(* POU PRG_STATION_LAYER3/FB_STATIONEN/FB_FUNCTION/FB_STATION, ST *)
FUNCTION_BLOCK FB_STATION
VAR_INPUT
	iConfigMachineType:INT;
	iConfigAxisType:INT;
	iConfigVisuNavigation:INT;
	rConfigMaxToolLength:REAL;
	xSafetyCircuitOn1:BOOL;
	xSafetyCircuitOn2:BOOL;
	T_ProcessImageData:ST_RETAIN_DATA_PROCESSIMAGE;
	T_Standard:ST_RETAIN_DATA;
	xActiveProcess:BOOL;
	iSelectToolTensionForce:INT;
END_VAR
VAR_IN_OUT
	TStation:ST_STATION;
	T_StartUp:ST_STARTUP;
END_VAR
VAR_OUTPUT
	xActive : BOOL :=FALSE;
	xStatusRdy : BOOL := FALSE;
	xStatusEnd : BOOL := FALSE;
	xStatusStop : BOOL := FALSE;
	xStatusRef : BOOL := FALSE;
	xError : BOOL := FALSE;
	iErrorNr : DINT :=0;
	iStatusFctNr : INT := 0;
	bActivePartNumber:BYTE;
	lrProcessToolFeederActualPosition:LREAL;
	lrProcessToolFeederSpeed:LREAL;
END_VAR
VAR
(* Pointer auf Actuatoren *)
	ptrTAxisToolLeft:POINTER TO ST_AXIS;
	ptrTAxisToolCenter:POINTER TO ST_AXIS;
	ptrTAxisToolRight:POINTER TO ST_AXIS;
	ptrTAxisToolFeeder:POINTER TO ST_AXIS;
	ptrTAxisGrindFeeder:POINTER TO ST_AXIS;
	ptrTCylToolTension:POINTER TO ST_CYLINDER;
(*22.12.2009: KFS {    *)
	ptrTCylToolLeftActive:POINTER TO ST_CYLINDER;
	ptrTCylToolRightActive:POINTER TO ST_CYLINDER;
	ptrTCylToolCenterActive:POINTER TO ST_CYLINDER;
	ptrTCylToolPrismaLeftActive:POINTER TO ST_CYLINDER;
	ptrTCylToolPrismaRightActive:POINTER TO ST_CYLINDER;
	ptrTToolFeederWorkLength:POINTER TO ST_CYLINDER;
(*22.12.2009: KFS }   *)
	ptrTFunction:POINTER TO ST_CTRL_FUNCTION;
	xSetEnableConfig: BOOL;
	iEnableConfigMachineType:INT;
	iTmpConfigMachineType:INT;
	iEnableConfigAxisType:INT;
	iTmpConfigAxisType:INT;
	iEnableConfigVisuNavigation:INT;
	iTmpConfigVisuNavigation:INT;
	rEnableConfigMaxToolLength:REAL;
	rTmpConfigMaxToolLength:REAL;
	xMicroRodActive: BOOL;
	xBeckhoffDriveActive: BOOL;
	xTmpStopFunction: BOOL;
	iStationFunctionNr: INT;
	xStartFunction: BOOL := FALSE;
	xTmpStart: BOOL := FALSE;
	xInitStart: BOOL := FALSE;
	xSetEnd: BOOL := FALSE;
	xInitError: BOOL := FALSE;
	xInitStop: BOOL := FALSE;
	xInitSetEnable: BOOL := FALSE;
	iStepEnable: INT := 0;
	xInitStep: BOOL := FALSE;
	iAxisFunctionNr: INT :=0;
	xInitDelEnable: BOOL := FALSE;
	xStationError: BOOL := FALSE;
	xStepError: BOOL;
	iStepError: INT;
	xTmpStationError: BOOL;
	xRdyDisableStation: BOOL;
	xReadyChkError: BOOL;
	xDontDeleteErrorFlag: BOOL;
	xSetError: BOOL;
(* Trigger *)
	fbFTrig: F_TRIG;
	fbRTrig: R_TRIG;
	xTmp: BOOL;
	diErrorNumber: DINT;
	iCountCycle: INT;
	xSecurityCircuitOn: BOOL;
	xSecurityCircuitOff: BOOL;
	iStepSecCircuit: INT;
	xInitSecCircuit: BOOL;
	TONCheckTimeOut: TON;
	xPowerSwitchedOn: BOOL;
	xChkConfigStation: BOOL;
	FBFctToolRotationTorqueStart: FB_FctToolRotationTorqueStart;
	FBFctToolRotationTorqueStop: FB_FctToolRotationTorqueStop;
	FBFctGrindFeedAbsRelPosition: FB_FctGrindFeedAbsRelPosition;
	FBFctSetAxisPosition: FB_FctSetAxisPosition;
	FBFctToolWorkingGeometry: FB_FctToolWorkingGeometry;
	FBFctToolWorkingGeometryMultiCycle: FB_FctToolWorkingGeometryMultiCycle;
	FBFctToolWorkingGroove: FB_FctToolWorkingGroove;
	FBFctToolCalibration: FB_FctToolCalibration;
	iMaxFunctionNr:INT:=20;
	(* 17.11.2010 KFS : iMaxFunctionNr:INT:=19*)
	FBFctToolFeedAbsRelPosition: FB_FctToolFeedAbsRelPosition;
	FBFctSwitchOnOffPowerSupply: FB_FctSwitchOnOffPowerSupply;
	(* 17.11.2010: KFS 	{	*)
	FBFctToolFeedMaxLenReference:FB_FctToolFeedMaxLenReference;
	(* 17.11.2010: KFS 	}	*)
	FBFctToolFeedReference: FB_FctToolFeedReference;
	xCheckAxisError: BOOL;
	xFirstTimeBooting: BOOL:=FALSE;
	FBFctStopAxisMovement: FB_FctStopAxisMovement;
	xAxisErrorActive: BOOL;
	xWaitSetError: BOOL;
	TONWaitSetError: TON;
	xForceHWError: BOOL;
	xCheckActiveFunction: BOOL;
	xForceResetAxis: BOOL;
	xReadyToQuitErr: BOOL;
	TONWaitReset: TON;
END_VAR
(****************************************************************************************************************************************************)
(***********                 This Functionblock manage all the station funtion and synchronizing of the Hardware                           ************)
(****************************************************************************************************************************************************)
xActive:=TStation.TControl.xActiveStation;
IF NOT(TStation.TControl.xActiveStation) THEN
	(*TStation:=TDeleteStationStruct;*)
	RETURN;
ELSE
	IF xSetEnableConfig THEN
		IF (iEnableConfigMachineType <> iConfigMachineType) THEN
			iTmpConfigMachineType:=iEnableConfigMachineType;
		ELSE
			iTmpConfigMachineType:=iConfigMachineType;
		END_IF;
		IF (iEnableConfigAxisType <> iConfigAxisType) THEN
			iTmpConfigAxisType:=iEnableConfigAxisType;
		ELSE
			iTmpConfigAxisType:=iConfigAxisType;
		END_IF;
		IF (iEnableConfigVisuNavigation <> iConfigVisuNavigation) THEN
			iTmpConfigVisuNavigation:=iEnableConfigVisuNavigation;
		ELSE
			iTmpConfigVisuNavigation:=iConfigVisuNavigation;
		END_IF;
		IF (rEnableConfigMaxToolLength <> rConfigMaxToolLength) THEN
			rTmpConfigMaxToolLength:=rEnableConfigMaxToolLength;
		ELSE
			rTmpConfigMaxToolLength:=rConfigMaxToolLength;
		END_IF;
		(*08.12.2010 KFS:	{	*)
		IF T_Station.xOverwriteMaxToolLength THEN
			rEnableConfigMaxToolLength:=rConfigMaxToolLength;
			rTmpConfigMaxToolLength:=rConfigMaxToolLength;
		END_IF;
		(*08.12.2010 KFS:	}	*)
	ELSE
		iTmpConfigMachineType:=iConfigMachineType;
		iTmpConfigAxisType:=iConfigAxisType;
		iTmpConfigVisuNavigation:=iConfigVisuNavigation;
		rTmpConfigMaxToolLength:=rConfigMaxToolLength;
	END_IF;
	(* Zuweisung der Datenstrukturen der Aktuatoren als Pointer *)
	ptrTAxisToolLeft:=ADR(TStation.THardware.TAxisToolLeft);
	ptrTAxisToolCenter:=ADR(TStation.THardware.TAxisToolCenter);
	ptrTAxisToolRight:=ADR(TStation.THardware.TAxisToolRight);
	ptrTAxisToolFeeder:=ADR(TStation.THardware.TAxisToolFeeder);
	ptrTAxisGrindFeeder:=ADR(TStation.THardware.TAxisGrindFeeder);
	ptrTCylToolTension:=ADR(TStation.THardware.TCylToolTension);
(*22.12.2009: KFS {    *)
	ptrTCylToolLeftActive:=ADR(TStation.THardware.TCylToolLeftActive);
	ptrTCylToolRightActive:=ADR(TStation.THardware.TCylToolRightActive);
	ptrTCylToolCenterActive:=ADR(TStation.THardware.TCylToolCenterActive);
	ptrTCylToolPrismaLeftActive:=ADR(TStation.THardware.TCylToolPrismaLeftActive);
	ptrTCylToolPrismaRightActive:=ADR(TStation.THardware.TCylToolPrismaRightActive);
	ptrTToolFeederWorkLength:=ADR(TStation.THardware.TToolFeederWorkLength);
(*22.12.2009: KFS }   *)
	ptrTFunction:=ADR(TStation.TCtrlFunction);
	IF (iConfigMachineType = 2) THEN
		xMicroRodActive:=TRUE;
	ELSE
		xMicroRodActive:=FALSE;
	END_IF;
	IF (iConfigAxisType = 2) THEN
		xBeckhoffDriveActive:=TRUE;
	ELSE
		xBeckhoffDriveActive:=FALSE;
	END_IF;
	IF xSafetyCircuitOn1 AND xSafetyCircuitOn2 THEN
		xPowerSwitchedOn:=TRUE;
	ELSE
		xPowerSwitchedOn:=FALSE;
	END_IF;
END_IF;
(******************************************************************************************************************************************)
(****************************				                  Status Part                                                            *****************************)
(******************************************************************************************************************************************)
xStatusRdy:=TStation.TControl.xRdy;
xStatusEnd:=TStation.TControl.xEnd;
xStatusStop:=xTmpStopFunction;
IF xMicroRodActive THEN
	TStation.TControl.xReferenced:=ptrTAxisToolFeeder^.T_CtrleSingle.xRef;
ELSE
	TStation.TControl.xReferenced:=TRUE;
END_IF;
xStatusRef:=TStation.TControl.xReferenced;
xError:= TStation.TControl.xError;
iErrorNr := TStation.TControl.diErrorNr;
iStatusFctNr:=iStationFunctionNr;
(******************************************************************************************************************************************)
(****************************				                Enable Part                                                            *****************************)
(******************************************************************************************************************************************)
(* Check Active of the Axis Drives *)
xTmp:=	(NOT(ptrTAxisToolLeft^.T_CtrleSingle.xErr) AND NOT(ptrTAxisToolLeft^.T_CtrleSingle.xDone)) OR
		(NOT(ptrTAxisToolCenter^.T_CtrleSingle.xErr) AND NOT(ptrTAxisToolCenter^.T_CtrleSingle.xDone) AND xMicroRodActive) OR
		(NOT(ptrTAxisToolRight^.T_CtrleSingle.xErr) AND NOT(ptrTAxisToolRight^.T_CtrleSingle.xDone)) OR
		(NOT(ptrTAxisToolFeeder^.T_CtrleSingle.xErr) AND NOT(ptrTAxisToolFeeder^.T_CtrleSingle.xDone)) OR
		(NOT(ptrTAxisGrindFeeder^.T_CtrleSingle.xErr) AND NOT(ptrTAxisGrindFeeder^.T_CtrleSingle.xDone));
fbFTrig(CLK:=TStation.TControl.xEnable);
IF fbFTrig.Q THEN
	xInitSetEnable:=FALSE;
	xInitDelEnable:=FALSE;
	xRdyDisableStation:=FALSE;
END_IF;
IF (fbFTrig.Q OR xInitDelEnable) THEN
	IF NOT(xInitDelEnable) OR fbFTrig.Q THEN
		xReadyChkError:=FALSE;
		TStation.TControl.xEnd:=FALSE;
		IF NOT(xDontDeleteErrorFlag) THEN
			TStation.TControl.xError:=FALSE;
		END_IF;
		xInitDelEnable:=TRUE;
		TStation.TControl.xRdy:=FALSE;
		iStepEnable:=100;
		iAxisFunctionNr:=1;
		iStationFunctionNr:=1;
		xInitStep:=FALSE;
	END_IF;
	CASE iStepEnable OF
		100:	IF NOT(xInitStep) THEN
				xInitStep:=TRUE;
				xSetEnableConfig:=FALSE;
				xStartFunction:=TRUE;
				ptrTFunction^.xReset:=TRUE;
			END_IF;
			IF NOT(ptrTFunction^.xReset) AND ptrTFunction^.xEnd THEN
				(* Alle Funktionen Resetten *)
				IF (iStationFunctionNr < iMaxFunctionNr) THEN
					iStationFunctionNr:=iStationFunctionNr + 1;
					ptrTFunction^.xReset:=TRUE;
				ELSE
					xInitStep:=FALSE;
					xStartFunction:=FALSE;
					iStepEnable:=200;
				END_IF;
			END_IF;
		200:	IF NOT(xInitStep) THEN
				xInitStep:=TRUE;
				IF TStation.TControl.xHardwareConfigError THEN
					TStation.TControl.xHardwareConfigError:=FALSE;
					TStation.TControl.xActiveHardware:=FALSE;
				ELSE
					xInitStep:=FALSE;
					iStepEnable:=300;
				END_IF;
				RETURN;
			END_IF;
			IF NOT(TStation.TControl.xError) OR xDontDeleteErrorFlag THEN
				TStation.TControl.xActiveHardware:=TRUE;
				xInitStep:=FALSE;
				iStepEnable:=300;
				RETURN;
			END_IF;
		300:	IF NOT(xInitStep) THEN	(* Alle Hardware Bausteine resetten *)
				xInitStep:=TRUE;
				ptrTCylToolTension^.T_CtrleCyl.xFBActiv:=FALSE;
				(*22.12.2009: KFS {    *)
				IF xMicroRodActive THEN
					ptrTCylToolLeftActive^.T_CtrleCyl.xFBActiv:=FALSE;
					ptrTCylToolRightActive^.T_CtrleCyl.xFBActiv:=FALSE;
					ptrTCylToolCenterActive^.T_CtrleCyl.xFBActiv:=FALSE;
					ptrTCylToolPrismaLeftActive^.T_CtrleCyl.xFBActiv:=FALSE;
					ptrTCylToolPrismaRightActive^.T_CtrleCyl.xFBActiv:=FALSE;
					ptrTToolFeederWorkLength^.T_CtrleCyl.xFBActiv:=FALSE;
				END_IF;
				(*22.12.2009: KFS }   *)
				IF xBeckhoffDriveActive THEN
					ptrTAxisToolLeft^.T_CtrleSingle.xReset:=TRUE;
					IF xMicroRodActive THEN
						ptrTAxisToolCenter^.T_CtrleSingle.xReset:=TRUE;
					END_IF;
					ptrTAxisToolRight^.T_CtrleSingle.xReset:=TRUE;
					ptrTAxisToolFeeder^.T_CtrleSingle.xReset:=TRUE;
					ptrTAxisGrindFeeder^.T_CtrleSingle.xReset:=TRUE;
				ELSE
					TStation.TControl.xResetHardware:=TRUE;
					iStepEnable:=399;
					RETURN;
				END_IF;
			END_IF;
			IF xTmp THEN
				RETURN;	(* Wait until all Drives finished *)
			END_IF;
			IF (NOT(ptrTAxisToolLeft^.T_CtrleSingle.xReset) AND ptrTAxisToolLeft^.T_CtrleSingle.xErr) OR
			    (((NOT(ptrTAxisToolCenter^.T_CtrleSingle.xReset) AND ptrTAxisToolCenter^.T_CtrleSingle.xErr AND xMicroRodActive) OR NOT(xMicroRodActive))) OR
			    (NOT(ptrTAxisToolRight^.T_CtrleSingle.xReset) AND ptrTAxisToolRight^.T_CtrleSingle.xErr) OR
			    (NOT(ptrTAxisToolFeeder^.T_CtrleSingle.xReset) AND ptrTAxisToolFeeder^.T_CtrleSingle.xErr)OR
			    (NOT(ptrTAxisGrindFeeder^.T_CtrleSingle.xReset) AND ptrTAxisGrindFeeder^.T_CtrleSingle.xErr) THEN
				xInitStep:=FALSE;
				iStepEnable:=400;
			END_IF;
			IF NOT(ptrTAxisToolLeft^.T_CtrleSingle.xReset) AND ptrTAxisToolLeft^.T_CtrleSingle.xDone AND
			    ((NOT(ptrTAxisToolCenter^.T_CtrleSingle.xReset) AND ptrTAxisToolCenter^.T_CtrleSingle.xDone AND xMicroRodActive) OR NOT(xMicroRodActive)) AND
			    NOT(ptrTAxisToolRight^.T_CtrleSingle.xReset) AND ptrTAxisToolRight^.T_CtrleSingle.xDone AND
			    NOT(ptrTAxisToolFeeder^.T_CtrleSingle.xReset) AND ptrTAxisToolFeeder^.T_CtrleSingle.xDone AND
			    NOT(ptrTAxisGrindFeeder^.T_CtrleSingle.xReset) AND ptrTAxisGrindFeeder^.T_CtrleSingle.xDone THEN
				TStation.TControl.xActiveHardware:=FALSE;
				xInitStep:=FALSE;
				xInitDelEnable:=FALSE;
				xSetEnd:=TRUE;
				xRdyDisableStation:=TRUE;
			END_IF;
		399:	IF NOT(TStation.TControl.xResetHardware) THEN
				TStation.TControl.xActiveHardware:=FALSE;
				xInitStep:=FALSE;
				xInitDelEnable:=FALSE;
				xSetEnd:=TRUE;
				xRdyDisableStation:=TRUE;
			END_IF;
		400:	IF NOT(xInitStep) THEN
				xInitStep:=TRUE;
				ptrTAxisToolLeft^.T_CtrleSingle.iFunction:=1;
				ptrTAxisToolLeft^.T_CtrleSingle.xExecute:=ptrTAxisToolLeft^.T_CtrleSingle.xErr;
				IF xMicroRodActive THEN
					ptrTAxisToolCenter^.T_CtrleSingle.iFunction:=1;
					ptrTAxisToolCenter^.T_CtrleSingle.xExecute:=ptrTAxisToolCenter^.T_CtrleSingle.xErr;
				END_IF;
				ptrTAxisToolRight^.T_CtrleSingle.iFunction:=1;
				ptrTAxisToolRight^.T_CtrleSingle.xExecute:=ptrTAxisToolRight^.T_CtrleSingle.xErr;
				ptrTAxisToolFeeder^.T_CtrleSingle.iFunction:=1;
				ptrTAxisToolFeeder^.T_CtrleSingle.xExecute:=ptrTAxisToolFeeder^.T_CtrleSingle.xErr;
				ptrTAxisGrindFeeder^.T_CtrleSingle.iFunction:=1;
				ptrTAxisGrindFeeder^.T_CtrleSingle.xExecute:=ptrTAxisGrindFeeder^.T_CtrleSingle.xErr;
			END_IF;
			IF xTmp THEN
				RETURN;	(* Wait until all Drives finished *)
			END_IF;
			IF NOT(ptrTAxisToolLeft^.T_CtrleSingle.xExecute) AND ptrTAxisToolLeft^.T_CtrleSingle.xErr AND
			    ((NOT(ptrTAxisToolCenter^.T_CtrleSingle.xExecute) AND ptrTAxisToolCenter^.T_CtrleSingle.xErr AND xMicroRodActive) OR NOT(xMicroRodActive)) AND
			    NOT(ptrTAxisToolRight^.T_CtrleSingle.xExecute) AND ptrTAxisToolRight^.T_CtrleSingle.xErr AND
			    NOT(ptrTAxisToolFeeder^.T_CtrleSingle.xExecute) AND ptrTAxisToolFeeder^.T_CtrleSingle.xErr AND
			    NOT(ptrTAxisGrindFeeder^.T_CtrleSingle.xExecute) AND ptrTAxisGrindFeeder^.T_CtrleSingle.xErr THEN
				xInitStep:=FALSE;
				iStepEnable:=500;
			END_IF;
			IF NOT(ptrTAxisToolLeft^.T_CtrleSingle.xExecute) AND ptrTAxisToolLeft^.T_CtrleSingle.xDone AND
			    ((NOT(ptrTAxisToolCenter^.T_CtrleSingle.xExecute) AND ptrTAxisToolCenter^.T_CtrleSingle.xDone AND xMicroRodActive) OR NOT(xMicroRodActive)) AND
			    NOT(ptrTAxisToolRight^.T_CtrleSingle.xExecute) AND ptrTAxisToolRight^.T_CtrleSingle.xDone AND
			    NOT(ptrTAxisToolFeeder^.T_CtrleSingle.xExecute) AND ptrTAxisToolFeeder^.T_CtrleSingle.xDone AND
			    NOT(ptrTAxisGrindFeeder^.T_CtrleSingle.xExecute) AND ptrTAxisGrindFeeder^.T_CtrleSingle.xDone THEN
				TStation.TControl.xActiveHardware:=FALSE;
				xInitStep:=FALSE;
				xInitDelEnable:=FALSE;
				xSetEnd:=TRUE;
				xRdyDisableStation:=TRUE;
			END_IF;
		500:	TStation.TControl.xActiveHardware:=FALSE;
			TStation.TControl.diErrorNr:=8000000 + 10;	(* Station Disable Fehlerhaft *)
			TStation.TControl.xError:=TRUE;
			xDontDeleteErrorFlag:=TRUE;
			xInitStep:=FALSE;
			xInitDelEnable:=FALSE;
			xSetEnd:=TRUE;
			xRdyDisableStation:=TRUE;
	END_CASE;
END_IF;
fbRTrig(CLK:=TStation.TControl.xEnable);
IF fbRTrig.Q THEN
	xInitSetEnable:=FALSE;
	xInitDelEnable:=FALSE;
END_IF;
IF (fbRTrig.Q OR xInitSetEnable) THEN
	IF NOT(fbRTrig.Q) AND xReadyChkError THEN
		IF xSetError OR ptrTAxisToolLeft^.T_CtrleSingle.xErr OR (ptrTAxisToolCenter^.T_CtrleSingle.xErr AND xMicroRodActive) OR
		     ptrTAxisToolRight^.T_CtrleSingle.xErr OR ptrTAxisToolFeeder^.T_CtrleSingle.xErr OR ptrTAxisGrindFeeder^.T_CtrleSingle.xErr THEN
			IF (xTmp OR (NOT(T_BoxID.T_Ctrle.xErr) AND NOT(T_BoxID.T_Ctrle.xDone))) AND NOT(xSetError) THEN
				RETURN;	(* Wait until all Actuators are not working *)
			END_IF;
			IF xSetError THEN
				xSetError:=FALSE;
				TStation.TControl.diErrorNr:=8000000 + diErrorNumber;
			ELSE
				ptrTAxisToolLeft^.T_CtrleSingle.xReset:=ptrTAxisToolLeft^.T_CtrleSingle.xErr;
				IF xMicroRodActive THEN
					ptrTAxisToolCenter^.T_CtrleSingle.xReset:=ptrTAxisToolCenter^.T_CtrleSingle.xErr;
				END_IF;
				ptrTAxisToolRight^.T_CtrleSingle.xReset:=ptrTAxisToolRight^.T_CtrleSingle.xErr;
				ptrTAxisToolFeeder^.T_CtrleSingle.xReset:=ptrTAxisToolFeeder^.T_CtrleSingle.xErr;
				ptrTAxisGrindFeeder^.T_CtrleSingle.xReset:=ptrTAxisGrindFeeder^.T_CtrleSingle.xErr;
				T_BoxID.T_Ctrle.xReset:=T_BoxID.T_Ctrle.xErr;
				IF ptrTAxisToolLeft^.T_CtrleSingle.xErr THEN TStation.TControl.diErrorNr:=1000000 + ptrTAxisToolLeft^.T_CtrleSingle.udiErrorID; END_IF;
				IF xMicroRodActive THEN
					IF ptrTAxisToolCenter^.T_CtrleSingle.xErr THEN TStation.TControl.diErrorNr:=2000000 + ptrTAxisToolCenter^.T_CtrleSingle.udiErrorID; END_IF;
				END_IF;
				IF ptrTAxisToolRight^.T_CtrleSingle.xErr THEN TStation.TControl.diErrorNr:=3000000 + ptrTAxisToolRight^.T_CtrleSingle.udiErrorID; END_IF;
				IF ptrTAxisToolFeeder^.T_CtrleSingle.xErr THEN TStation.TControl.diErrorNr:=4000000 + ptrTAxisToolFeeder^.T_CtrleSingle.udiErrorID; END_IF;
				IF ptrTAxisGrindFeeder^.T_CtrleSingle.xErr THEN TStation.TControl.diErrorNr:=5000000 + ptrTAxisGrindFeeder^.T_CtrleSingle.udiErrorID; END_IF;
				IF T_BoxID.T_Ctrle.xErr THEN TStation.TControl.diErrorNr:=7000000 + T_BoxID.T_Ctrle.udiErrorID; END_IF;
			END_IF;
			TStation.TControl.xEnable:=FALSE;
			TStation.TControl.xError:=TRUE;
			xDontDeleteErrorFlag:=TRUE;
			RETURN;
		END_IF;
	END_IF;
	IF NOT(xInitSetEnable) OR fbRTrig.Q THEN
		xSetEnd:=FALSE;
		xInitSetEnable:=TRUE;
		TStation.TControl.xRdy:=FALSE;
		TStation.TControl.xEnd:=FALSE;
		TStation.TControl.xError:=FALSE;
		TStation.TControl.diErrorNr:=0;
		iStepEnable:=100;
		iAxisFunctionNr:=1;
		iStationFunctionNr:=1;
		xSetEnableConfig:=FALSE;
		xInitStep:=FALSE;
		RETURN;
	END_IF;
	CASE iStepEnable OF
		100:	IF NOT(xRdyDisableStation) THEN
				iStepEnable:=110;
				RETURN;
			END_IF;
			IF NOT(xInitStep) THEN
				xInitStep:=TRUE;
				xStartFunction:=TRUE;
				ptrTFunction^.xReset:=TRUE;
				(* Initialisierung der HW *)
				TStation.TControl.xActiveHardware:=TRUE;
				TStation.T_MachineConfig.iConfigMachineType:=iConfigMachineType;
				TStation.T_MachineConfig.iConfigAxisType:=iConfigAxisType;
				TStation.T_MachineConfig.iConfigVisuNavigation:=iConfigVisuNavigation;
				TStation.T_MachineConfig.rConfigMaxToolLength:=rConfigMaxToolLength;
				(* Initialisierung der Aktuatoren *)

			(* Config Cyl ToolTension *)
				ptrTCylToolTension^.T_CtrleCyl.xFBActiv:=TRUE;
				ptrTCylToolTension^.T_Config.xActivState:=TRUE;
				(*22.12.2009: KFS {    *)
				IF xMicroRodActive THEN
				(* Config Cyl ToolLeftActive*)
					ptrTCylToolLeftActive^.T_CtrleCyl.xFBActiv:=TRUE;
					ptrTCylToolLeftActive^.T_Config.xActivState:=TRUE;
				(* Config Cyl ToolRightActive*)
					ptrTCylToolRightActive^.T_CtrleCyl.xFBActiv:=TRUE;
					ptrTCylToolRightActive^.T_Config.xActivState:=TRUE;
				(* Config Cyl ToolCenterActive*)
					ptrTCylToolCenterActive^.T_CtrleCyl.xFBActiv:=TRUE;
					ptrTCylToolCenterActive^.T_Config.xActivState:=TRUE;
				(* Config Cyl ToolPrismaLeftActive*)
					ptrTCylToolPrismaLeftActive^.T_CtrleCyl.xFBActiv:=TRUE;
					ptrTCylToolPrismaLeftActive^.T_Config.xActivState:=TRUE;
				(* Config Cyl ToolPrismaRightActive*)
					ptrTCylToolPrismaRightActive^.T_CtrleCyl.xFBActiv:=TRUE;
					ptrTCylToolPrismaRightActive^.T_Config.xActivState:=TRUE;
				(* Config Cyl ToolWorkLength*)
					ptrTToolFeederWorkLength^.T_CtrleCyl.xFBActiv:=TRUE;
					ptrTToolFeederWorkLength^.T_Config.xActivState:=TRUE;
				END_IF;
				(*22.12.2009: KFS }   *)
			(* Config ToolLeft Axis *)
				ptrTAxisToolLeft^.T_Config_Gen.iTyp:=1;
				ptrTAxisToolLeft^.T_Config_Gen.iMachineType:=iConfigMachineType;
				ptrTAxisToolLeft^.T_Config_ObjFileValue.xSWLimitNeg:=FALSE;
				ptrTAxisToolLeft^.T_Config_ObjFileValue.xSWLimitPos:=FALSE;
				ptrTAxisToolLeft^.T_Config_ObjFileValue.xHWLimitNeg:=FALSE;
				ptrTAxisToolLeft^.T_Config_ObjFileValue.xHWLimitPos:=FALSE;
			(* Config ToolCenter Axis *)
				IF xMicroRodActive THEN
					ptrTAxisToolCenter^.T_Config_Gen.iTyp:=2;
					ptrTAxisToolCenter^.T_Config_Gen.iMachineType:=iConfigMachineType;
					ptrTAxisToolCenter^.T_Config_ObjFileValue.xSWLimitNeg:=FALSE;
					ptrTAxisToolCenter^.T_Config_ObjFileValue.xSWLimitPos:=FALSE;
					ptrTAxisToolCenter^.T_Config_ObjFileValue.xHWLimitNeg:=FALSE;
					ptrTAxisToolCenter^.T_Config_ObjFileValue.xHWLimitPos:=FALSE;
				END_IF;
			(* Config ToolRight Axis *)
				ptrTAxisToolRight^.T_Config_Gen.iTyp:=3;
				ptrTAxisToolRight^.T_Config_Gen.iMachineType:=iConfigMachineType;
				ptrTAxisToolRight^.T_Config_ObjFileValue.xSWLimitNeg:=FALSE;
				ptrTAxisToolRight^.T_Config_ObjFileValue.xSWLimitPos:=FALSE;
				ptrTAxisToolRight^.T_Config_ObjFileValue.xHWLimitNeg:=FALSE;
				ptrTAxisToolRight^.T_Config_ObjFileValue.xHWLimitPos:=FALSE;
			(* Config ToolFeeder Axis *)
				ptrTAxisToolFeeder^.T_Config_Gen.iTyp:=4;
				ptrTAxisToolFeeder^.T_Config_Gen.iMachineType:=iConfigMachineType;
				IF xMicroRodActive THEN
					ptrTAxisToolFeeder^.T_Config_ObjFileValue.xSWLimitNeg:=FALSE;
					ptrTAxisToolFeeder^.T_Config_ObjFileValue.xSWLimitPos:=FALSE;
				   	ptrTAxisToolFeeder^.T_Config_ObjFileValue.xHWLimitNeg:=TRUE;
					ptrTAxisToolFeeder^.T_Config_ObjFileValue.xHWLimitPos:=TRUE;
				ELSE
					ptrTAxisToolFeeder^.T_Config_ObjFileValue.xSWLimitNeg:=FALSE;
					ptrTAxisToolFeeder^.T_Config_ObjFileValue.xSWLimitPos:=FALSE;
					ptrTAxisToolFeeder^.T_Config_ObjFileValue.xHWLimitNeg:=FALSE;
					ptrTAxisToolFeeder^.T_Config_ObjFileValue.xHWLimitPos:=FALSE;
				END_IF;
			(* Config GrindFeeder Axis *)
				ptrTAxisGrindFeeder^.T_Config_Gen.iTyp:=5;
				ptrTAxisGrindFeeder^.T_Config_Gen.iMachineType:=iConfigMachineType;
				ptrTAxisGrindFeeder^.T_Config_ObjFileValue.xSWLimitNeg:=TRUE;
				ptrTAxisGrindFeeder^.T_Config_ObjFileValue.xSWLimitPos:=TRUE;
				ptrTAxisGrindFeeder^.T_Config_ObjFileValue.xHWLimitNeg:=FALSE;
				ptrTAxisGrindFeeder^.T_Config_ObjFileValue.xHWLimitPos:=FALSE;
			END_IF;
			IF NOT(ptrTFunction^.xReset) AND ptrTFunction^.xEnd THEN
				(* Alle Funktionen Resetten *)
				IF (iStationFunctionNr < iMaxFunctionNr) THEN
					iStationFunctionNr:=iStationFunctionNr + 1;
					ptrTFunction^.xReset:=TRUE;
				ELSE
					xInitStep:=FALSE;
					xStartFunction:=FALSE;
					iStepEnable:=200;
				END_IF;
			END_IF;
		110:	IF NOT(xInitStep) THEN
				xInitStep:=TRUE;
				IF TStation.TControl.xHardwareConfigError THEN
					TStation.TControl.xHardwareConfigError:=FALSE;
					TStation.TControl.xActiveHardware:=FALSE;
				ELSE
					xRdyDisableStation:=TRUE;
					xInitStep:=FALSE;
					iStepEnable:=100;
				END_IF;
				RETURN;
			END_IF;
			IF NOT(TStation.TControl.xError) THEN
				TStation.TControl.xActiveHardware:=TRUE;
				xRdyDisableStation:=TRUE;
				xInitStep:=FALSE;
				iStepEnable:=100;
				RETURN;
			END_IF;
		200:	IF NOT(xInitStep) THEN
				xInitStep:=TRUE;
				ptrTCylToolTension^.T_CtrleCyl.xReset:=TRUE;
				(*22.12.2009: KFS {    *)
				IF xMicroRodActive THEN
					ptrTCylToolLeftActive^.T_CtrleCyl.xReset:=TRUE;
					ptrTCylToolRightActive^.T_CtrleCyl.xReset:=TRUE;
					ptrTCylToolCenterActive^.T_CtrleCyl.xReset:=TRUE;
					ptrTCylToolPrismaLeftActive^.T_CtrleCyl.xReset:=TRUE;
					ptrTCylToolPrismaRightActive^.T_CtrleCyl.xReset:=TRUE;
					ptrTToolFeederWorkLength^.T_CtrleCyl.xReset:=TRUE;
				END_IF;
				(*22.12.2009: KFS }   *)
				ptrTAxisToolLeft^.T_CtrleSingle.xReset:=TRUE;
				IF xMicroRodActive THEN
					ptrTAxisToolCenter^.T_CtrleSingle.xReset:=TRUE;
				END_IF;
				ptrTAxisToolRight^.T_CtrleSingle.xReset:=TRUE;
				ptrTAxisToolFeeder^.T_CtrleSingle.xReset:=TRUE;
				ptrTAxisGrindFeeder^.T_CtrleSingle.xReset:=TRUE;
			END_IF;
			IF NOT(ptrTAxisToolLeft^.T_CtrleSingle.xReset) AND NOT(ptrTAxisToolCenter^.T_CtrleSingle.xReset) AND ((NOT(ptrTAxisToolRight^.T_CtrleSingle.xReset) AND xMicroRodActive) OR NOT(xMicroRodActive)) AND
			     NOT(ptrTAxisToolFeeder^.T_CtrleSingle.xReset) AND NOT(ptrTAxisGrindFeeder^.T_CtrleSingle.xReset) THEN
				xInitStep:=FALSE;
				IF NOT(xBeckhoffDriveActive) THEN
					iStepEnable:=300;
				ELSE
					iStepEnable:=500;
				END_IF;
			END_IF;
		300:	IF NOT(xInitStep) THEN
				xInitStep:=TRUE;
				ptrTAxisToolLeft^.T_CtrleSingle.lrAcceleration:=T_Standard.T_TeachINToolLeft.rAcceleration;
				ptrTAxisToolLeft^.T_CtrleSingle.lrDecceleration:=T_Standard.T_TeachINToolLeft.rDeceleration;
				ptrTAxisToolCenter^.T_CtrleSingle.lrAcceleration:=T_Standard.T_TeachINToolCenter.rAcceleration;
				ptrTAxisToolCenter^.T_CtrleSingle.lrDecceleration:=T_Standard.T_TeachINToolCenter.rDeceleration;
				ptrTAxisToolRight^.T_CtrleSingle.lrAcceleration:=T_Standard.T_TeachINToolRight.rAcceleration;
				ptrTAxisToolRight^.T_CtrleSingle.lrDecceleration:=T_Standard.T_TeachINToolRight.rDeceleration;
				ptrTAxisToolFeeder^.T_CtrleSingle.lrAcceleration:=T_Standard.T_TeachINToolFeeder.rAcceleration;
				ptrTAxisToolFeeder^.T_CtrleSingle.lrDecceleration:=T_Standard.T_TeachINToolFeeder.rDeceleration;
				ptrTAxisGrindFeeder^.T_CtrleSingle.lrAcceleration:=T_Standard.T_TeachINGrindFeeder.rAcceleration;
				ptrTAxisGrindFeeder^.T_CtrleSingle.lrDecceleration:=T_Standard.T_TeachINGrindFeeder.rDeceleration;
				ptrTAxisToolLeft^.T_Config_Gen.sFileNamePDOMapping:='PDOMapping_ToolLeft';
				ptrTAxisToolLeft^.T_CtrleSingle.iFunction:=22;
				ptrTAxisToolLeft^.T_CtrleSingle.xExecute:=TRUE;
				IF xMicroRodActive THEN
					ptrTAxisToolCenter^.T_Config_Gen.sFileNamePDOMapping:='PDOMapping_ToolCenter';
					ptrTAxisToolCenter^.T_CtrleSingle.iFunction:=22;
					ptrTAxisToolCenter^.T_CtrleSingle.xExecute:=TRUE;
				END_IF;
				ptrTAxisToolRight^.T_Config_Gen.sFileNamePDOMapping:='PDOMapping_ToolRight';
				ptrTAxisToolRight^.T_CtrleSingle.iFunction:=22;
				ptrTAxisToolRight^.T_CtrleSingle.xExecute:=TRUE;
				ptrTAxisToolFeeder^.T_Config_Gen.sFileNamePDOMapping:='PDOMapping_ToolFeeder';
				ptrTAxisToolFeeder^.T_CtrleSingle.iFunction:=22;
				ptrTAxisToolFeeder^.T_CtrleSingle.xExecute:=TRUE;
				ptrTAxisGrindFeeder^.T_Config_Gen.sFileNamePDOMapping:='PDOMapping_GrindFeeder';
				ptrTAxisGrindFeeder^.T_CtrleSingle.iFunction:=22;
				ptrTAxisGrindFeeder^.T_CtrleSingle.xExecute:=TRUE;
				iCountCycle:=0;
			END_IF;
			iCountCycle:=iCountCycle + 1;
			IF (iCountCycle >= 50) THEN
				xReadyChkError:=TRUE;	(* 50 SPS Zyklen warten bis die Übewachung der HW Error freigeschaltet werden kann *)
			END_IF;
			IF xTmp THEN
				RETURN;	(* Wait until all Drives finished *)
			END_IF;
			IF NOT(ptrTAxisToolLeft^.T_CtrleSingle.xExecute) AND ptrTAxisToolLeft^.T_CtrleSingle.xDone AND
			    ((NOT(ptrTAxisToolCenter^.T_CtrleSingle.xExecute) AND ptrTAxisToolCenter^.T_CtrleSingle.xDone AND xMicroRodActive) OR NOT(xMicroRodActive)) AND
			    NOT(ptrTAxisToolRight^.T_CtrleSingle.xExecute) AND ptrTAxisToolRight^.T_CtrleSingle.xDone AND
			    NOT(ptrTAxisToolFeeder^.T_CtrleSingle.xExecute) AND ptrTAxisToolFeeder^.T_CtrleSingle.xDone AND
			    NOT(ptrTAxisGrindFeeder^.T_CtrleSingle.xExecute) AND ptrTAxisGrindFeeder^.T_CtrleSingle.xDone THEN
				xReadyChkError:=TRUE;
				xInitStep:=FALSE;
				iStepEnable:=400;
			END_IF;
		400:	IF NOT(xInitStep) THEN
				xInitStep:=TRUE;
				ptrTAxisToolLeft^.T_CtrleSingle.iFunction:=23;
				ptrTAxisToolLeft^.T_CtrleSingle.xExecute:=TRUE;
				IF xMicroRodActive THEN
					ptrTAxisToolCenter^.T_CtrleSingle.iFunction:=23;
					ptrTAxisToolCenter^.T_CtrleSingle.xExecute:=TRUE;
				END_IF;
				ptrTAxisToolRight^.T_CtrleSingle.iFunction:=23;
				ptrTAxisToolRight^.T_CtrleSingle.xExecute:=TRUE;
				ptrTAxisToolFeeder^.T_CtrleSingle.iFunction:=23;
				ptrTAxisToolFeeder^.T_CtrleSingle.xExecute:=TRUE;
				ptrTAxisGrindFeeder^.T_CtrleSingle.iFunction:=23;
				ptrTAxisGrindFeeder^.T_CtrleSingle.xExecute:=TRUE;
			END_IF;
			IF xTmp THEN
				RETURN;	(* Wait until all Drives finished *)
			END_IF;
			IF NOT(ptrTAxisToolLeft^.T_CtrleSingle.xExecute) AND ptrTAxisToolLeft^.T_CtrleSingle.xDone AND
			    ((NOT(ptrTAxisToolCenter^.T_CtrleSingle.xExecute) AND ptrTAxisToolCenter^.T_CtrleSingle.xDone AND xMicroRodActive) OR NOT(xMicroRodActive)) AND
			    NOT(ptrTAxisToolRight^.T_CtrleSingle.xExecute) AND ptrTAxisToolRight^.T_CtrleSingle.xDone AND
			    NOT(ptrTAxisToolFeeder^.T_CtrleSingle.xExecute) AND ptrTAxisToolFeeder^.T_CtrleSingle.xDone AND
			    NOT(ptrTAxisGrindFeeder^.T_CtrleSingle.xExecute) AND ptrTAxisGrindFeeder^.T_CtrleSingle.xDone THEN
				xInitStep:=FALSE;
				iStepEnable:=500;
			END_IF;
		500:	IF NOT(xInitStep) THEN
				xInitStep:=TRUE;
				ptrTAxisToolLeft^.T_CtrleSingle.iFunction:=1;
				ptrTAxisToolLeft^.T_CtrleSingle.xExecute:=TRUE;
				IF xMicroRodActive THEN
					ptrTAxisToolCenter^.T_CtrleSingle.iFunction:=1;
					ptrTAxisToolCenter^.T_CtrleSingle.xExecute:=TRUE;
				END_IF;
				ptrTAxisToolRight^.T_CtrleSingle.iFunction:=1;
				ptrTAxisToolRight^.T_CtrleSingle.xExecute:=TRUE;
				ptrTAxisToolFeeder^.T_CtrleSingle.iFunction:=1;
				ptrTAxisToolFeeder^.T_CtrleSingle.xExecute:=TRUE;
				ptrTAxisGrindFeeder^.T_CtrleSingle.iFunction:=1;
				ptrTAxisGrindFeeder^.T_CtrleSingle.xExecute:=TRUE;
			END_IF;
			IF NOT(ptrTAxisToolLeft^.T_CtrleSingle.xExecute) AND ptrTAxisToolLeft^.T_CtrleSingle.xDone AND
			    ((NOT(ptrTAxisToolCenter^.T_CtrleSingle.xExecute) AND ptrTAxisToolCenter^.T_CtrleSingle.xDone AND xMicroRodActive) OR NOT(xMicroRodActive)) AND
			    NOT(ptrTAxisToolRight^.T_CtrleSingle.xExecute) AND ptrTAxisToolRight^.T_CtrleSingle.xDone AND
			    NOT(ptrTAxisToolFeeder^.T_CtrleSingle.xExecute) AND ptrTAxisToolFeeder^.T_CtrleSingle.xDone AND
			    NOT(ptrTAxisGrindFeeder^.T_CtrleSingle.xExecute) AND ptrTAxisGrindFeeder^.T_CtrleSingle.xDone THEN
				xInitStep:=FALSE;
				iStepEnable:=600;
			END_IF;
		600:	IF NOT(xInitStep) THEN	(* Read Axis Parameter File *)
				xInitStep:=TRUE;
				ptrTAxisToolLeft^.T_Config_Gen.sDeviceFileName:='EcoStep23S21_ToolLeft';
				ptrTAxisToolLeft^.T_CtrleSingle.iFunction:=2;
				ptrTAxisToolLeft^.T_CtrleSingle.xExecute:=TRUE;
				IF xMicroRodActive THEN
					ptrTAxisToolCenter^.T_Config_Gen.sDeviceFileName:='EcoStep23S21_ToolCenter';
					ptrTAxisToolCenter^.T_CtrleSingle.iFunction:=2;
					ptrTAxisToolCenter^.T_CtrleSingle.xExecute:=TRUE;
				END_IF;
				ptrTAxisToolRight^.T_Config_Gen.sDeviceFileName:='EcoStep23S21_ToolRight';
				ptrTAxisToolRight^.T_CtrleSingle.iFunction:=2;
				ptrTAxisToolRight^.T_CtrleSingle.xExecute:=TRUE;
				ptrTAxisToolFeeder^.T_Config_Gen.sDeviceFileName:='EcoStep23S21_ToolFeeder';
				ptrTAxisToolFeeder^.T_CtrleSingle.iFunction:=2;
				ptrTAxisToolFeeder^.T_CtrleSingle.xExecute:=TRUE;
				ptrTAxisGrindFeeder^.T_Config_Gen.sDeviceFileName:='EcoStep23S21_GrindFeeder';
				ptrTAxisGrindFeeder^.T_CtrleSingle.iFunction:=2;
				ptrTAxisGrindFeeder^.T_CtrleSingle.xExecute:=TRUE;
			END_IF;
			IF NOT(ptrTAxisToolLeft^.T_CtrleSingle.xExecute) AND ptrTAxisToolLeft^.T_CtrleSingle.xDone AND
			    ((NOT(ptrTAxisToolCenter^.T_CtrleSingle.xExecute) AND ptrTAxisToolCenter^.T_CtrleSingle.xDone AND xMicroRodActive) OR NOT(xMicroRodActive)) AND
			    NOT(ptrTAxisToolRight^.T_CtrleSingle.xExecute) AND ptrTAxisToolRight^.T_CtrleSingle.xDone AND
			    NOT(ptrTAxisToolFeeder^.T_CtrleSingle.xExecute) AND ptrTAxisToolFeeder^.T_CtrleSingle.xDone AND
			    NOT(ptrTAxisGrindFeeder^.T_CtrleSingle.xExecute) AND ptrTAxisGrindFeeder^.T_CtrleSingle.xDone THEN
				xInitStep:=FALSE;
				iStepEnable:=700;
			END_IF;
		700:	IF NOT(xInitStep) THEN	(* Read Axis Parameter File *)
				xInitStep:=TRUE;
				ptrTAxisToolLeft^.T_CtrleSingle.iFunction:=21;
				ptrTAxisToolLeft^.T_CtrleSingle.xExecute:=TRUE;
				IF xMicroRodActive THEN
					ptrTAxisToolCenter^.T_CtrleSingle.iFunction:=21;
					ptrTAxisToolCenter^.T_CtrleSingle.xExecute:=TRUE;
				END_IF;
				ptrTAxisToolRight^.T_CtrleSingle.iFunction:=21;
				ptrTAxisToolRight^.T_CtrleSingle.xExecute:=TRUE;
				ptrTAxisToolFeeder^.T_CtrleSingle.iFunction:=21;
				ptrTAxisToolFeeder^.T_CtrleSingle.xExecute:=TRUE;
				ptrTAxisGrindFeeder^.T_CtrleSingle.iFunction:=21;
				ptrTAxisGrindFeeder^.T_CtrleSingle.xExecute:=TRUE;
			END_IF;
			IF NOT(ptrTAxisToolLeft^.T_CtrleSingle.xExecute) AND ptrTAxisToolLeft^.T_CtrleSingle.xDone AND
			    ((NOT(ptrTAxisToolCenter^.T_CtrleSingle.xExecute) AND ptrTAxisToolCenter^.T_CtrleSingle.xDone AND xMicroRodActive) OR NOT(xMicroRodActive)) AND
			    NOT(ptrTAxisToolRight^.T_CtrleSingle.xExecute) AND ptrTAxisToolRight^.T_CtrleSingle.xDone AND
			    NOT(ptrTAxisToolFeeder^.T_CtrleSingle.xExecute) AND ptrTAxisToolFeeder^.T_CtrleSingle.xDone AND
			    NOT(ptrTAxisGrindFeeder^.T_CtrleSingle.xExecute) AND ptrTAxisGrindFeeder^.T_CtrleSingle.xDone THEN
				xInitStep:=FALSE;
				IF NOT(xBeckhoffDriveActive) THEN
					iStepEnable:=1000;
				ELSE
					iStepEnable:=800;
				END_IF;
			END_IF;
		800:	IF NOT(xInitStep) THEN
				IF NOT(T_BoxID.T_Ctrle.xLocked) THEN
					xInitStep:=TRUE;
					(* Box ID-->Beckhoff drive *)
					T_BoxID.T_Ctrle.iMachineType:=iConfigMachineType;
					T_BoxID.T_Servo_ToolLeft.sBoxName:='AX25xx_Slide_St1';
					T_BoxID.T_Servo_ToolLeft.sDeviceName:='AX25xx_Slide_St1';
					T_BoxID.T_Servo_ToolLeft.xDeviceOption:=TRUE;
					T_BoxID.T_Servo_ToolCenter.sBoxName:='AX25xx_Slide_St1';
					T_BoxID.T_Servo_ToolCenter.sDeviceName:='AX25xx_Slide_St1';
					T_BoxID.T_Servo_ToolCenter.xDeviceOption:=TRUE;
					T_BoxID.T_Servo_ToolRight.sBoxName:='AX25xx_Slide_St1';
					T_BoxID.T_Servo_ToolRight.sDeviceName:='AX25xx_Slide_St1';
					T_BoxID.T_Servo_ToolRight.xDeviceOption:=TRUE;
					T_BoxID.T_Servo_ToolFeeder.sBoxName:='AX25xx_Slide_St1';
					T_BoxID.T_Servo_ToolFeeder.sDeviceName:='AX25xx_Slide_St1';
					T_BoxID.T_Servo_ToolFeeder.xDeviceOption:=TRUE;
					T_BoxID.T_Servo_GrindFeeder.sBoxName:='AX25xx_Slide_St1';
					T_BoxID.T_Servo_GrindFeeder.sDeviceName:='AX25xx_Slide_St1';
					T_BoxID.T_Servo_GrindFeeder.xDeviceOption:=TRUE;
					T_BoxID.T_Ctrle.xLocked:=TRUE;
					T_BoxID.T_Ctrle.xExecute:=TRUE;
				END_IF;
				RETURN;
			END_IF;
			IF NOT(T_BoxID.T_Ctrle.xExecute) AND T_BoxID.T_Ctrle.xDone AND T_BoxID.T_Ctrle.xLocked THEN
				T_BoxID.T_Ctrle.xLocked:=FALSE;
				xInitStep:=FALSE;
				iStepEnable:=900;
			END_IF;
		900:	IF NOT(xInitStep) THEN
				xInitStep:=TRUE;
				IF (T_BoxID.T_Servo_ToolLeft.wAddrBox = 0) OR (T_BoxID.T_Servo_ToolLeft.wAddrBox <> ptrTAxisToolLeft^.T_Config_Gen.udiNC_TaskIdxGrp) THEN
					xSetError:=TRUE;
					diErrorNumber:=16#F201;	(* ToolLeft-->Falsche Konfiguration oder Achse nicht vorhanden *)
					RETURN;
				ELSIF ((T_BoxID.T_Servo_ToolCenter.wAddrBox = 0) OR (T_BoxID.T_Servo_ToolCenter.wAddrBox <> ptrTAxisToolCenter^.T_Config_Gen.udiNC_TaskIdxGrp)) AND xMicroRodActive THEN
					xSetError:=TRUE;
					diErrorNumber:=16#F202;	(* ToolCenter-->Falsche Konfiguration oder Achse nicht vorhanden *)
					RETURN;
				ELSIF (T_BoxID.T_Servo_ToolRight.wAddrBox = 0) OR (T_BoxID.T_Servo_ToolRight.wAddrBox <> ptrTAxisToolRight^.T_Config_Gen.udiNC_TaskIdxGrp) THEN
					xSetError:=TRUE;
					diErrorNumber:=16#F203;	(* ToolRight-->Falsche Konfiguration oder Achse nicht vorhanden *)
					RETURN;
				ELSIF (T_BoxID.T_Servo_ToolFeeder.wAddrBox = 0) OR (T_BoxID.T_Servo_ToolFeeder.wAddrBox <> ptrTAxisToolFeeder^.T_Config_Gen.udiNC_TaskIdxGrp) THEN
					xSetError:=TRUE;
					diErrorNumber:=16#F204;	(* ToolFeeder-->Falsche Konfiguration oder Achse nicht vorhanden *)
					RETURN;
				ELSIF (T_BoxID.T_Servo_GrindFeeder.wAddrBox = 0) OR (T_BoxID.T_Servo_GrindFeeder.wAddrBox <> ptrTAxisGrindFeeder^.T_Config_Gen.udiNC_TaskIdxGrp) THEN
					xSetError:=TRUE;
					diErrorNumber:=16#F205;	(* GrindFeeder-->Falsche Konfiguration oder Achse nicht vorhanden *)
					RETURN;
				ELSE
				(* Achsenparameterisierung erfolgreich *)
					;
				END_IF;
				xInitStep:=FALSE;
				iStepEnable:=1100;
			END_IF;
		(* Read Axis Firmware Information *)
		1000:IF NOT(xInitStep) THEN
				xInitStep:=TRUE;
				ptrTAxisToolLeft^.T_CtrleSingle.iFunction:=27;
				ptrTAxisToolLeft^.T_CtrleSingle.xExecute:=TRUE;
				IF xMicroRodActive THEN
					ptrTAxisToolCenter^.T_CtrleSingle.iFunction:=27;
					ptrTAxisToolCenter^.T_CtrleSingle.xExecute:=TRUE;
				END_IF;
				ptrTAxisToolRight^.T_CtrleSingle.iFunction:=27;
				ptrTAxisToolRight^.T_CtrleSingle.xExecute:=TRUE;
				ptrTAxisToolFeeder^.T_CtrleSingle.iFunction:=27;
				ptrTAxisToolFeeder^.T_CtrleSingle.xExecute:=TRUE;
				ptrTAxisGrindFeeder^.T_CtrleSingle.iFunction:=27;
				ptrTAxisGrindFeeder^.T_CtrleSingle.xExecute:=TRUE;
			END_IF;
			IF NOT(ptrTAxisToolLeft^.T_CtrleSingle.xExecute) AND ptrTAxisToolLeft^.T_CtrleSingle.xDone AND
			    ((NOT(ptrTAxisToolCenter^.T_CtrleSingle.xExecute) AND ptrTAxisToolCenter^.T_CtrleSingle.xDone AND xMicroRodActive) OR NOT(xMicroRodActive)) AND
			    NOT(ptrTAxisToolRight^.T_CtrleSingle.xExecute) AND ptrTAxisToolRight^.T_CtrleSingle.xDone AND
			    NOT(ptrTAxisToolFeeder^.T_CtrleSingle.xExecute) AND ptrTAxisToolFeeder^.T_CtrleSingle.xDone AND
			    NOT(ptrTAxisGrindFeeder^.T_CtrleSingle.xExecute) AND ptrTAxisGrindFeeder^.T_CtrleSingle.xDone THEN
				xInitStep:=FALSE;
				iStepEnable:=1100;
			END_IF;
		1100:IF NOT(xInitStep) THEN
				xInitStep:=TRUE;
				ptrTAxisToolLeft^.T_CtrleSingle.iFunction:=4;
				ptrTAxisToolLeft^.T_CtrleSingle.xExecute:=TRUE;
				IF xMicroRodActive THEN
					ptrTAxisToolCenter^.T_CtrleSingle.iFunction:=4;
					ptrTAxisToolCenter^.T_CtrleSingle.xExecute:=TRUE;
				END_IF;
				ptrTAxisToolRight^.T_CtrleSingle.iFunction:=4;
				ptrTAxisToolRight^.T_CtrleSingle.xExecute:=TRUE;
				ptrTAxisToolFeeder^.T_CtrleSingle.iFunction:=4;
				ptrTAxisToolFeeder^.T_CtrleSingle.xExecute:=TRUE;
				ptrTAxisGrindFeeder^.T_CtrleSingle.iFunction:=4;
				ptrTAxisGrindFeeder^.T_CtrleSingle.xExecute:=TRUE;
			END_IF;
			IF NOT(ptrTAxisToolLeft^.T_CtrleSingle.xExecute) AND ptrTAxisToolLeft^.T_CtrleSingle.xDone AND
			    ((NOT(ptrTAxisToolCenter^.T_CtrleSingle.xExecute) AND ptrTAxisToolCenter^.T_CtrleSingle.xDone AND xMicroRodActive) OR NOT(xMicroRodActive)) AND
			    NOT(ptrTAxisToolRight^.T_CtrleSingle.xExecute) AND ptrTAxisToolRight^.T_CtrleSingle.xDone AND
			    NOT(ptrTAxisToolFeeder^.T_CtrleSingle.xExecute) AND ptrTAxisToolFeeder^.T_CtrleSingle.xDone AND
			    NOT(ptrTAxisGrindFeeder^.T_CtrleSingle.xExecute) AND ptrTAxisGrindFeeder^.T_CtrleSingle.xDone THEN
				xInitStep:=FALSE;
				iStepEnable:=1200;
			END_IF;
		1200:IF NOT(xInitStep) THEN
				xInitStep:=TRUE;
				ptrTAxisToolLeft^.T_CtrleSingle.iFunction:=3;
				ptrTAxisToolLeft^.T_CtrleSingle.xExecute:=TRUE;
				IF xMicroRodActive THEN
					ptrTAxisToolCenter^.T_CtrleSingle.iFunction:=3;
					ptrTAxisToolCenter^.T_CtrleSingle.xExecute:=TRUE;
				END_IF;
				ptrTAxisToolRight^.T_CtrleSingle.iFunction:=3;
				ptrTAxisToolRight^.T_CtrleSingle.xExecute:=TRUE;
				ptrTAxisToolFeeder^.T_CtrleSingle.iFunction:=3;
				ptrTAxisToolFeeder^.T_CtrleSingle.xExecute:=TRUE;
				ptrTAxisGrindFeeder^.T_CtrleSingle.iFunction:=3;
				ptrTAxisGrindFeeder^.T_CtrleSingle.xExecute:=TRUE;
			END_IF;
			IF NOT(ptrTAxisToolLeft^.T_CtrleSingle.xExecute) AND ptrTAxisToolLeft^.T_CtrleSingle.xDone AND
			    ((NOT(ptrTAxisToolCenter^.T_CtrleSingle.xExecute) AND ptrTAxisToolCenter^.T_CtrleSingle.xDone AND xMicroRodActive) OR NOT(xMicroRodActive)) AND
			    NOT(ptrTAxisToolRight^.T_CtrleSingle.xExecute) AND ptrTAxisToolRight^.T_CtrleSingle.xDone AND
			    NOT(ptrTAxisToolFeeder^.T_CtrleSingle.xExecute) AND ptrTAxisToolFeeder^.T_CtrleSingle.xDone AND
			    NOT(ptrTAxisGrindFeeder^.T_CtrleSingle.xExecute) AND ptrTAxisGrindFeeder^.T_CtrleSingle.xDone THEN
				IF NOT(xFirstTimeBooting) THEN
					xFirstTimeBooting:=TRUE;
					iStepEnable:=1300;
				ELSE
					iStepEnable:=1400;
				END_IF;
				xInitStep:=FALSE;
			END_IF;
		(* Set the Position of the GrindFeeder on the Settled ToolDiameter, but only on the first time on booting of the machine *)
		1300:IF NOT(xInitStep) THEN
				xInitStep:=TRUE;
				ptrTAxisGrindFeeder^.T_CtrleSingle.rSetPosition:=T_ProcessImageData.T_ProcessPara.rToolDiameterProcess;
				ptrTAxisGrindFeeder^.T_CtrleSingle.iFunction:=11;
				ptrTAxisGrindFeeder^.T_CtrleSingle.xExecute:=TRUE;
			END_IF;
			IF NOT(ptrTAxisGrindFeeder^.T_CtrleSingle.xExecute) AND ptrTAxisGrindFeeder^.T_CtrleSingle.xDone THEN
				xInitStep:=FALSE;
				iStepEnable:=1400;
			END_IF;
		(* Set the SW Limit position for the GrindFeeder Axis *)
		1400:IF NOT(xInitStep) THEN
				xInitStep:=TRUE;
				ptrTAxisGrindFeeder^.T_CtrleSingle.lrSWNegLimitSwitch:=T_ProcessImageData.T_PrismPara.rToolDiameterMin;
				ptrTAxisGrindFeeder^.T_CtrleSingle.lrSWPosLimitSwitch:=T_ProcessImageData.T_PrismPara.rToolDiameterMax + T_Standard.T_TeachINGrindFeeder.rOffsetSWPosEndSwitch;
				ptrTAxisGrindFeeder^.T_CtrleSingle.iFunction:=28;
				ptrTAxisGrindFeeder^.T_CtrleSingle.xExecute:=TRUE;
			END_IF;
			IF NOT(ptrTAxisGrindFeeder^.T_CtrleSingle.xExecute) AND ptrTAxisGrindFeeder^.T_CtrleSingle.xDone THEN
				xInitStep:=FALSE;
				IF NOT(xMicroRodActive) THEN
					(* Only for MicroWire activate the ToolTension *)
					iStepEnable:=1500;
				ELSE
					iStepEnable:=1600;
				END_IF;
			END_IF;
		1500:IF NOT(xInitStep) THEN
				xInitStep:=TRUE;
				ptrTCylToolTension^.T_CtrleCyl.iFunction:=2;
				ptrTCylToolTension^.T_CtrleCyl.T_AnalogCylinder.rForceIn:=T_ProcessImageData.T_ProcessPara.rToolTensionProcess;
				ptrTCylToolTension^.T_CtrleCyl.xExecute:=TRUE;
			END_IF;
			IF NOT(ptrTCylToolTension^.T_CtrleCyl.xExecute) AND ptrTCylToolTension^.T_CtrleCyl.xDone THEN
				xInitStep:=FALSE;
				iStepEnable:=1600;
			END_IF;
		1600:xReadyChkError:=FALSE;
			xInitStep:=FALSE;
			xSetEnableConfig:=TRUE;
			iEnableConfigMachineType:=iConfigMachineType;
			iEnableConfigAxisType:=iConfigAxisType;
			iEnableConfigVisuNavigation:=iConfigVisuNavigation;
			rEnableConfigMaxToolLength:=rConfigMaxToolLength;
			xInitSetEnable:=FALSE;
			TStation.TControl.xRdy:=TRUE;
			xSetEnd:=TRUE;
	END_CASE;
END_IF;
(******************************************************************************************************************************************)
(****************************				       Security Circuit Switch ON/OFF                                          *****************************)
(******************************************************************************************************************************************)
IF (TStation.TControl.xSecurityCircuitOn OR TStation.TControl.xSecurityCircuitOff OR xSecurityCircuitOn OR xSecurityCircuitOff) AND NOT(xInitSetEnable) AND NOT(xInitDelEnable) THEN
	IF NOT(xSecurityCircuitOn) AND NOT(xSecurityCircuitOff) THEN
		xSecurityCircuitOn:=TStation.TControl.xSecurityCircuitOn;
		xSecurityCircuitOff:=TStation.TControl.xSecurityCircuitOff;
		iStepSecCircuit:=1;
		xInitSecCircuit:=FALSE;
		TStation.TControl.xRdy:=FALSE;
		TStation.TControl.xEnd:=FALSE;
		TONCheckTimeOut(IN:=FALSE);
	END_IF;
	IF xSecurityCircuitOn THEN
		IF TStation.TControl.xSecurityCircuitOff THEN
			TStation.TControl.xSecurityCircuitOn:=FALSE;
			xSecurityCircuitOn:=FALSE;
		END_IF;
	END_IF;
	IF xSecurityCircuitOff THEN
		IF TStation.TControl.xSecurityCircuitOn THEN
			TStation.TControl.xSecurityCircuitOff:=FALSE;
			xSecurityCircuitOff:=FALSE;
		END_IF;
	END_IF;
	TONCheckTimeOut(IN:=TRUE,PT:=T#0.5s);
	xCheckAxisError:=FALSE;
	IF TONCheckTimeOut.Q THEN
		IF ptrTAxisToolLeft^.T_CtrleSingle.xErr THEN
			ptrTAxisToolLeft^.T_CtrleSingle.iFunction:=1;
			ptrTAxisToolLeft^.T_CtrleSingle.xExecute:=TRUE;
			xCheckAxisError:=TRUE;
		END_IF;
		IF xMicroRodActive THEN
			IF ptrTAxisToolCenter^.T_CtrleSingle.xErr THEN
				ptrTAxisToolCenter^.T_CtrleSingle.iFunction:=1;
				ptrTAxisToolCenter^.T_CtrleSingle.xExecute:=TRUE;
				xCheckAxisError:=TRUE;
			END_IF;
		END_IF;
		IF ptrTAxisToolRight^.T_CtrleSingle.xErr THEN
			ptrTAxisToolRight^.T_CtrleSingle.iFunction:=1;
			ptrTAxisToolRight^.T_CtrleSingle.xExecute:=TRUE;
			xCheckAxisError:=TRUE;
		END_IF;
		IF ptrTAxisToolFeeder^.T_CtrleSingle.xErr THEN
			ptrTAxisToolFeeder^.T_CtrleSingle.iFunction:=1;
			ptrTAxisToolFeeder^.T_CtrleSingle.xExecute:=TRUE;
			xCheckAxisError:=TRUE;
		END_IF;
		IF ptrTAxisGrindFeeder^.T_CtrleSingle.xErr THEN
			ptrTAxisGrindFeeder^.T_CtrleSingle.iFunction:=1;
			ptrTAxisGrindFeeder^.T_CtrleSingle.xExecute:=TRUE;
			xCheckAxisError:=TRUE;
		END_IF;
		TStation.TControl.xRdy:=TRUE;
		IF xCheckAxisError THEN
			TStation.TControl.xSecurityCircuitOn:=FALSE;
			TStation.TControl.xSecurityCircuitOff:=FALSE;
			xSecurityCircuitOn:=FALSE;
			xSecurityCircuitOff:=FALSE;
			iStepSecCircuit:=1;
			xInitSecCircuit:=FALSE;
			xSetEnd:=TRUE;
			RETURN;
		END_IF;
	END_IF;
	CASE iStepSecCircuit OF
	1:	IF NOT(xInitSecCircuit) THEN
			xInitSecCircuit:=TRUE;
			ptrTFunction^.xReset:=TRUE;
			iStationFunctionNr:=1;
			xStartFunction:=TRUE;
		END_IF;
		IF NOT(ptrTFunction^.xReset) AND ptrTFunction^.xEnd THEN
			(* Alle Funktionen Resetten *)
			IF (iStationFunctionNr < iMaxFunctionNr) THEN
				iStationFunctionNr:=iStationFunctionNr + 1;
				ptrTFunction^.xReset:=TRUE;
			ELSE
				xInitSecCircuit:=FALSE;
				iStepSecCircuit:=10;
				xStartFunction:=FALSE;
			END_IF;
		END_IF;
	10:	IF NOT(xInitSecCircuit) THEN
			xInitSecCircuit:=TRUE;
			ptrTAxisToolLeft^.T_CtrleSingle.xReset:=TRUE;
			IF xMicroRodActive THEN
				ptrTAxisToolCenter^.T_CtrleSingle.xReset:=TRUE;
			END_IF;
			ptrTAxisToolRight^.T_CtrleSingle.xReset:=TRUE;
			ptrTAxisToolFeeder^.T_CtrleSingle.xReset:=TRUE;
			ptrTAxisGrindFeeder^.T_CtrleSingle.xReset:=TRUE;
		END_IF;
		IF NOT(ptrTAxisToolLeft^.T_CtrleSingle.xReset) AND ((NOT(ptrTAxisToolCenter^.T_CtrleSingle.xReset) AND xMicroRodActive) OR NOT(xMicroRodActive)) AND NOT(ptrTAxisToolRight^.T_CtrleSingle.xReset) AND
		    NOT(ptrTAxisToolFeeder^.T_CtrleSingle.xReset) AND NOT(ptrTAxisGrindFeeder^.T_CtrleSingle.xReset) THEN
			xInitSecCircuit:=FALSE;
			iStepSecCircuit:=20;
		END_IF;
	20:	IF NOT(xInitSecCircuit) THEN
			xInitSecCircuit:=TRUE;
			ptrTAxisToolLeft^.T_CtrleSingle.iFunction:=1;
			ptrTAxisToolLeft^.T_CtrleSingle.xExecute:=TRUE;
			IF xMicroRodActive THEN
				ptrTAxisToolCenter^.T_CtrleSingle.iFunction:=1;
				ptrTAxisToolCenter^.T_CtrleSingle.xExecute:=TRUE;
			END_IF;
			ptrTAxisToolRight^.T_CtrleSingle.iFunction:=1;
			ptrTAxisToolRight^.T_CtrleSingle.xExecute:=TRUE;
			ptrTAxisToolFeeder^.T_CtrleSingle.iFunction:=1;
			ptrTAxisToolFeeder^.T_CtrleSingle.xExecute:=TRUE;
			ptrTAxisGrindFeeder^.T_CtrleSingle.iFunction:=1;
			ptrTAxisGrindFeeder^.T_CtrleSingle.xExecute:=TRUE;
		END_IF;
		IF NOT(ptrTAxisToolLeft^.T_CtrleSingle.xExecute) AND ptrTAxisToolLeft^.T_CtrleSingle.xDone AND
		    ((NOT(ptrTAxisToolCenter^.T_CtrleSingle.xExecute) AND ptrTAxisToolCenter^.T_CtrleSingle.xDone AND xMicroRodActive) OR NOT(xMicroRodActive)) AND
		    NOT(ptrTAxisToolRight^.T_CtrleSingle.xExecute) AND ptrTAxisToolRight^.T_CtrleSingle.xDone AND
		    NOT(ptrTAxisToolFeeder^.T_CtrleSingle.xExecute) AND ptrTAxisToolFeeder^.T_CtrleSingle.xDone AND
		    NOT(ptrTAxisGrindFeeder^.T_CtrleSingle.xExecute) AND ptrTAxisGrindFeeder^.T_CtrleSingle.xDone THEN
			xInitSecCircuit:=FALSE;
			iStepSecCircuit:=30;
		END_IF;
	30:	IF NOT(xInitSecCircuit) THEN
			xInitSecCircuit:=TRUE;
			(* Resetten der Aktuatoren *)
			ptrTCylToolTension^.T_CtrleCyl.xReset:=TRUE;
			(*22.12.2009: KFS {    *)
			IF xMicroRodActive THEN
				ptrTCylToolLeftActive^.T_CtrleCyl.xReset:=TRUE;
				ptrTCylToolRightActive^.T_CtrleCyl.xReset:=TRUE;
				ptrTCylToolCenterActive^.T_CtrleCyl.xReset:=TRUE;
				ptrTCylToolPrismaLeftActive^.T_CtrleCyl.xReset:=TRUE;
				ptrTCylToolPrismaRightActive^.T_CtrleCyl.xReset:=TRUE;
			END_IF;
			(*22.12.2009: KFS }   *)
		END_IF;
		IF NOT(ptrTCylToolTension^.T_CtrleCyl.xReset) AND ptrTCylToolTension^.T_CtrleCyl.xDone AND
		     ( NOT(xMicroRodActive) OR
		         ( NOT(ptrTCylToolLeftActive^.T_CtrleCyl.xReset) AND ptrTCylToolLeftActive^.T_CtrleCyl.xDone AND
		           NOT(ptrTCylToolRightActive^.T_CtrleCyl.xReset) AND ptrTCylToolRightActive^.T_CtrleCyl.xDone AND
		           NOT(ptrTCylToolCenterActive^.T_CtrleCyl.xReset) AND ptrTCylToolCenterActive^.T_CtrleCyl.xDone AND
 		           NOT(ptrTCylToolPrismaLeftActive^.T_CtrleCyl.xReset) AND ptrTCylToolPrismaLeftActive^.T_CtrleCyl.xDone AND
                              NOT(ptrTCylToolPrismaRightActive^.T_CtrleCyl.xReset) AND ptrTCylToolPrismaRightActive^.T_CtrleCyl.xDone )  )  THEN
			xInitSecCircuit:=FALSE;
			IF xSecurityCircuitOn THEN
				iStepSecCircuit:=40;
			ELSE
				iStepSecCircuit:=50;
			END_IF;
		END_IF;
	40:	IF NOT(xInitSecCircuit) THEN
				xInitSecCircuit:=TRUE;
				ptrTAxisToolLeft^.T_CtrleSingle.iFunction:=3;
				ptrTAxisToolLeft^.T_CtrleSingle.xExecute:=TRUE;
				IF xMicroRodActive THEN
					ptrTAxisToolCenter^.T_CtrleSingle.iFunction:=3;
					ptrTAxisToolCenter^.T_CtrleSingle.xExecute:=TRUE;
				END_IF;
				ptrTAxisToolRight^.T_CtrleSingle.iFunction:=3;
				ptrTAxisToolRight^.T_CtrleSingle.xExecute:=TRUE;
				ptrTAxisToolFeeder^.T_CtrleSingle.iFunction:=3;
				ptrTAxisToolFeeder^.T_CtrleSingle.xExecute:=TRUE;
				ptrTAxisGrindFeeder^.T_CtrleSingle.iFunction:=3;
				ptrTAxisGrindFeeder^.T_CtrleSingle.xExecute:=TRUE;
				IF NOT(xMicroRodActive) THEN
					ptrTCylToolTension^.T_CtrleCyl.iFunction:=2;
					IF (iSelectToolTensionForce < 2) THEN
						ptrTCylToolTension^.T_CtrleCyl.T_AnalogCylinder.rForceIn:=T_ProcessImageData.T_ProcessPara.rToolTensionProcess;
					END_IF;
					IF (iSelectToolTensionForce > 1) THEN
						ptrTCylToolTension^.T_CtrleCyl.T_AnalogCylinder.rForceIn:=T_Standard.T_Cyl_ToolTension.rForce;
					END_IF
					ptrTCylToolTension^.T_CtrleCyl.xExecute:=TRUE;
				END_IF;
			END_IF;
			IF NOT(ptrTAxisToolLeft^.T_CtrleSingle.xExecute) AND ptrTAxisToolLeft^.T_CtrleSingle.xDone AND
			    ((NOT(ptrTAxisToolCenter^.T_CtrleSingle.xExecute) AND ptrTAxisToolCenter^.T_CtrleSingle.xDone AND xMicroRodActive) OR NOT(xMicroRodActive)) AND
			    NOT(ptrTAxisToolRight^.T_CtrleSingle.xExecute) AND ptrTAxisToolRight^.T_CtrleSingle.xDone AND
			    NOT(ptrTAxisToolFeeder^.T_CtrleSingle.xExecute) AND ptrTAxisToolFeeder^.T_CtrleSingle.xDone AND
			    NOT(ptrTAxisGrindFeeder^.T_CtrleSingle.xExecute) AND ptrTAxisGrindFeeder^.T_CtrleSingle.xDone AND
			    ((NOT(ptrTCylToolTension^.T_CtrleCyl.xExecute) AND ptrTCylToolTension^.T_CtrleCyl.xDone AND NOT(xMicroRodActive)) OR xMicroRodActive) THEN
				xInitSecCircuit:=FALSE;
				iStepSecCircuit:=50;
			END_IF;
	50:	TStation.TControl.xRdy:=TRUE;
		TStation.TControl.xSecurityCircuitOn:=FALSE;
		TStation.TControl.xSecurityCircuitOff:=FALSE;
		xSecurityCircuitOn:=FALSE;
		xSecurityCircuitOff:=FALSE;
		iStepSecCircuit:=1;
		xInitSecCircuit:=FALSE;
		xSetEnd:=TRUE;
	END_CASE;
ELSE
	TStation.TControl.xSecurityCircuitOn:=FALSE;
	TStation.TControl.xSecurityCircuitOff:=FALSE;
	xSecurityCircuitOn:=FALSE;
	xSecurityCircuitOff:=FALSE;
	iStepSecCircuit:=1;
	xInitSecCircuit:=FALSE;
	TONCheckTimeOut(IN:=FALSE);
END_IF;
(******************************************************************************************************************************************)
(****************************				         Error Controlling Part                                                  *****************************)
(******************************************************************************************************************************************)
IF xActiveProcess THEN
	IF (ptrTAxisToolLeft^.T_CtrleSingle.xErr OR (ptrTAxisToolCenter^.T_CtrleSingle.xErr AND xMicroRodActive) OR ptrTAxisToolRight^.T_CtrleSingle.xErr OR
              ptrTAxisToolFeeder^.T_CtrleSingle.xErr OR ptrTAxisGrindFeeder^.T_CtrleSingle.xErr) AND NOT(xWaitSetError) THEN
		xWaitSetError:=TRUE;
		TONWaitSetError(IN:=FALSE);
	END_IF;
	IF xWaitSetError THEN
		TONWaitSetError(IN:=TRUE,PT:=T#50ms);
		IF TONWaitSetError.Q THEN
			xForceHWError:=TRUE;
		END_IF;
	END_IF;
ELSE
	xWaitSetError:=FALSE;
	xForceHWError:=FALSE;
	TONWaitSetError(IN:=FALSE);
END_IF;
IF xStationError OR xForceHWError OR (ptrTFunction^.xError AND TStation.TControl.xRdy AND NOT(xSetEnd)) THEN
	IF NOT(xInitError) THEN
		xForceHWError:=FALSE;
		xStationError:=TRUE;
		xTmpStationError:=TRUE;
		xInitError:=TRUE;
		xAxisErrorActive:=FALSE;
		TStation.TControl.diErrorNr:=0;
		IF ptrTAxisToolLeft^.T_CtrleSingle.xErr THEN
			TStation.TControl.diErrorNr:=1000000 + ptrTAxisToolLeft^.T_CtrleSingle.udiErrorID;
			ptrTAxisToolLeft^.T_CtrleSingle.iFunction:=1;
			ptrTAxisToolLeft^.T_CtrleSingle.xExecute:=TRUE;
			xAxisErrorActive:=TRUE;
		END_IF;
		IF xMicroRodActive THEN
			IF ptrTAxisToolCenter^.T_CtrleSingle.xErr THEN
				TStation.TControl.diErrorNr:=2000000 + ptrTAxisToolCenter^.T_CtrleSingle.udiErrorID;
				ptrTAxisToolCenter^.T_CtrleSingle.iFunction:=1;
				ptrTAxisToolCenter^.T_CtrleSingle.xExecute:=TRUE;
				xAxisErrorActive:=TRUE;
			END_IF;
		END_IF;
		IF ptrTAxisToolRight^.T_CtrleSingle.xErr THEN
			TStation.TControl.diErrorNr:=3000000 + ptrTAxisToolRight^.T_CtrleSingle.udiErrorID;
			ptrTAxisToolRight^.T_CtrleSingle.iFunction:=1;
			ptrTAxisToolRight^.T_CtrleSingle.xExecute:=TRUE;
			xAxisErrorActive:=TRUE;
		END_IF;
		IF ptrTAxisToolFeeder^.T_CtrleSingle.xErr THEN
			TStation.TControl.diErrorNr:=4000000 + ptrTAxisToolFeeder^.T_CtrleSingle.udiErrorID;
			ptrTAxisToolFeeder^.T_CtrleSingle.iFunction:=1;
			ptrTAxisToolFeeder^.T_CtrleSingle.xExecute:=TRUE;
			xAxisErrorActive:=TRUE;
		END_IF;
		IF ptrTAxisGrindFeeder^.T_CtrleSingle.xErr THEN
			TStation.TControl.diErrorNr:=5000000 + ptrTAxisGrindFeeder^.T_CtrleSingle.udiErrorID;
			ptrTAxisGrindFeeder^.T_CtrleSingle.iFunction:=1;
			ptrTAxisGrindFeeder^.T_CtrleSingle.xExecute:=TRUE;
			xAxisErrorActive:=TRUE;
		END_IF;
		IF ptrTCylToolTension^.T_CtrleCyl.xErr THEN
			TStation.TControl.diErrorNr:=6000000 + ptrTCylToolTension^.T_CtrleCyl.udiErrorID;
			ptrTCylToolTension^.T_CtrleCyl.xReset:=TRUE;
		END_IF;
		IF (TStation.TControl.diErrorNr = 0) THEN	(* General Error-->No Hardware Error  7000 - 7999*)
			TStation.TControl.diErrorNr:=8000000 + ptrTFunction^.iErrorNr;
		END_IF;
		ptrTFunction^.xQuitErr:=NOT(ptrTFunction^.xEnd) AND ptrTFunction^.xError;
		IF NOT(ptrTFunction^.xQuitErr) AND NOT(ptrTFunction^.xEnd) THEN
			xForceResetAxis:=TRUE;
			ptrTFunction^.xReset:=TRUE;
		END_IF;
		TONWaitReset(IN:=FALSE);
	END_IF;
	IF (ptrTFunction^.xEnd OR xForceResetAxis) AND xTmpStationError THEN
		IF NOT(ptrTAxisToolLeft^.T_CtrleSingle.xErr) AND ((NOT(ptrTAxisToolCenter^.T_CtrleSingle.xErr) AND xMicroRodActive) OR NOT(xMicroRodActive)) AND
		     NOT(ptrTAxisToolRight^.T_CtrleSingle.xErr) AND NOT(ptrTAxisToolFeeder^.T_CtrleSingle.xErr) AND NOT(ptrTAxisGrindFeeder^.T_CtrleSingle.xErr) THEN
			TStation.TControl.xError:=TRUE;
			xForceResetAxis:=FALSE;
		END_IF;
		TONWaitReset(IN:=TRUE,PT:=T#100ms);
		IF TONWaitReset.Q THEN
			IF xAxisErrorActive THEN
				T_StartUp.T_Ctrle.xSetSecurityStateON:=TRUE;
			END_IF;
			xStepError:=FALSE;
			xStartFunction:=FALSE;
			xTmpStationError:=FALSE;
			xReadyToQuitErr:=TRUE;
		END_IF;
	END_IF;
	IF TStation.TControl.xQuitError AND NOT(ptrTFunction^.xQuitErr) AND xReadyToQuitErr THEN
		xInitError:=FALSE;
		TStation.TControl.xQuitError:=FALSE;
		xSetEnd:=TRUE;
	END_IF;
END_IF;
(******************************************************************************************************************************************)
(****************************				         Main Controlling Part                                                  *****************************)
(******************************************************************************************************************************************)
IF (TStation.TControl.xStart OR xTmpStart) AND TStation.TControl.xRdy AND NOT(xSetEnd) THEN
	IF NOT(xInitStart) THEN
		xInitStart:=TRUE;
		xTmpStart:=TRUE;
		TStation.TControl.xStart:=FALSE;
		TStation.TControl.xEnd:=FALSE;
		ptrTFunction^.xStart:=TRUE;
		xStartFunction:=TRUE;
		iStationFunctionNr:=TStation.TControl.iFunctNr;
		TStation.TControl.xAbord:=FALSE;
	END_IF;
	IF TStation.TControl.xStop THEN
		IF NOT(xInitStop) THEN
			xInitStop:=TRUE;
			ptrTFunction^.xStop:=TRUE;
		END_IF;
		IF NOT(ptrTFunction^.xStop) THEN
			xInitStop:=FALSE;
			TStation.TControl.xStop:=FALSE;
			xTmpStopFunction:=TRUE;
		END_IF;
	END_IF;
	IF TStation.TControl.xStart AND xTmpStopFunction AND NOT(ptrTFunction^.xAbord) THEN
		TStation.TControl.xStart:=FALSE;
		xTmpStopFunction:=FALSE;
		ptrTFunction^.xStart:=TRUE;
	END_IF;
	IF TStation.TControl.xAbord AND xTmpStopFunction THEN
		TStation.TControl.xAbord:=FALSE;
		xTmpStopFunction:=FALSE;
		ptrTFunction^.xStart:=FALSE;
		ptrTFunction^.xAbord:=TRUE;
	END_IF;
	IF NOT(ptrTFunction^.xStart) AND ptrTFunction^.xEnd AND NOT(xStationError) THEN
		xTmpStart:=FALSE;
		xInitStart:=FALSE;
		xSetEnd:=TRUE;
	END_IF;
END_IF;
(******************************************************************************************************************************************)
(****************************				   Check Configuration Station Part                                 *****************************)
(******************************************************************************************************************************************)
IF (xStartFunction OR xChkConfigStation) AND xSetEnableConfig THEN
	IF NOT(xChkConfigStation) THEN
		IF (iEnableConfigMachineType <> iConfigMachineType) OR (iEnableConfigAxisType <> iConfigAxisType) OR (iEnableConfigVisuNavigation <> iConfigVisuNavigation) OR (rEnableConfigMaxToolLength <> rConfigMaxToolLength)  THEN
			xChkConfigStation:=TRUE;
			ptrTFunction^.xStop:=NOT(ptrTFunction^.xEnd);
			IF ptrTFunction^.xEnd THEN
				ptrTFunction^.xStart:=FALSE;
			END_IF;
		END_IF;
	END_IF;
	IF xChkConfigStation THEN
		IF ptrTFunction^.xEnd THEN
			IF (iEnableConfigMachineType <> iConfigMachineType) THEN
				ptrTFunction^.iErrorNr:=7001;	(* Error-->Config Machine Type changed *)
			END_IF;
			IF (iEnableConfigAxisType <> iConfigAxisType) THEN
				ptrTFunction^.iErrorNr:=7002;	(* Error-->Config Axis Type changed *)
			END_IF;
			IF (iEnableConfigVisuNavigation <> iConfigVisuNavigation) THEN
				TStation.TControl.diErrorNr:=7003;	(* Error-->Config Visu Navigation changed *)
			END_IF;
			IF (rEnableConfigMaxToolLength <> rConfigMaxToolLength) THEN
				TStation.TControl.diErrorNr:=7004;	(* Error-->Config Max Tool Length changed *)
			END_IF;
			xStartFunction:=FALSE;
			xChkConfigStation:=FALSE;
			xStationError:=TRUE;
			RETURN;
		END_IF;
	END_IF;
END_IF;
(******************************************************************************************************************************************)
(****************************				              Funktionen                                                               *****************************)
(******************************************************************************************************************************************)
IF xStartFunction AND NOT(xSetEnd) THEN
	IF (iStationFunctionNr = 1) THEN
		FBFctToolFeedReference(	xMicroRodActive:= xMicroRodActive,
								xBeckhoffDriveActive:= xBeckhoffDriveActive,
								xSafetyCircuitOn:= xSafetyCircuitOn1 AND xSafetyCircuitOn2,
								T_Standard:= T_Standard,
								xStart:= ptrTFunction^.xStart,
								xReset:=ptrTFunction^.xReset,
								xStop:= ptrTFunction^.xStop,
								xQuitErr:= ptrTFunction^.xQuitErr,
								xAbord:= ptrTFunction^.xAbord,
								TAxisToolFeeder:= ptrTAxisToolFeeder^,
								xEnd=>ptrTFunction^.xEnd,
								xError=>ptrTFunction^.xError,
								iErrorNr=>ptrTFunction^.iErrorNr);
	END_IF;
	IF (iStationFunctionNr = 2) THEN
		FBFctToolRotationTorqueStart(	xMicroRodActive:= xMicroRodActive,
									xBeckhoffDriveActive:= xBeckhoffDriveActive,
									xSafetyCircuitOn:=xSafetyCircuitOn1 AND xSafetyCircuitOn2,
									xStart:= ptrTFunction^.xStart,
									xReset:=ptrTFunction^.xReset,
									xStop:= ptrTFunction^.xStop,
									xQuitErr:= ptrTFunction^.xQuitErr,
									xAbord:= ptrTFunction^.xAbord,
									TAxisToolLeft:= ptrTAxisToolLeft^,
									TAxisToolCenter:= ptrTAxisToolCenter^,
									TAxisToolRight:=ptrTAxisToolRight^,
									TAxisToolFeeder:=ptrTAxisToolFeeder^,
									xEnd=>ptrTFunction^.xEnd,
									xError=>ptrTFunction^.xError,
									iErrorNr=>ptrTFunction^.iErrorNr);
	END_IF;
	IF (iStationFunctionNr = 3) THEN
		FBFctToolRotationTorqueStop(	xMicroRodActive:= xMicroRodActive,
									xBeckhoffDriveActive:= xBeckhoffDriveActive,
									xSafetyCircuitOn:=xSafetyCircuitOn1 AND xSafetyCircuitOn2,
									xStart:= ptrTFunction^.xStart,
									xReset:=ptrTFunction^.xReset,
									xStop:= ptrTFunction^.xStop,
									xQuitErr:= ptrTFunction^.xQuitErr,
									xAbord:= ptrTFunction^.xAbord,
									TAxisToolLeft:= ptrTAxisToolLeft^,
									TAxisToolCenter:= ptrTAxisToolCenter^,
									TAxisToolRight:=ptrTAxisToolRight^,
									TAxisToolFeeder:=ptrTAxisToolFeeder^,
									xEnd=>ptrTFunction^.xEnd,
									xError=>ptrTFunction^.xError,
									iErrorNr=>ptrTFunction^.iErrorNr);
	END_IF;
	IF (iStationFunctionNr = 4) OR (iStationFunctionNr = 5) THEN
		FBFctGrindFeedAbsRelPosition(	xMicroRodActive:= xMicroRodActive,
										xBeckhoffDriveActive:= xBeckhoffDriveActive,
										xSafetyCircuitOn:= xSafetyCircuitOn1 AND xSafetyCircuitOn2,
										iFunctionNr:= iStationFunctionNr,
										xStart:= ptrTFunction^.xStart,
										xReset:=ptrTFunction^.xReset,
										xStop:= ptrTFunction^.xStop,
										xQuitErr:= ptrTFunction^.xQuitErr,
										xAbord:= ptrTFunction^.xAbord,
										TAxisGrindFeeder:= ptrTAxisGrindFeeder^,
										xEnd=>ptrTFunction^.xEnd,
										xError=>ptrTFunction^.xError,
										iErrorNr=>ptrTFunction^.iErrorNr);
	END_IF;
	IF (iStationFunctionNr >= 6) AND (iStationFunctionNr <= 10) THEN
		FBFctSetAxisPosition(	xMicroRodActive:= xMicroRodActive,
							xBeckhoffDriveActive:= xBeckhoffDriveActive,
							xSafetyCircuitOn:= xSafetyCircuitOn1 AND xSafetyCircuitOn2,
							iFunctionNr:= iStationFunctionNr,
							xStart:= ptrTFunction^.xStart,
							xReset:=ptrTFunction^.xReset,
							xStop:= ptrTFunction^.xStop,
							xQuitErr:= ptrTFunction^.xQuitErr,
							xAbord:= ptrTFunction^.xAbord,
							TAxisToolLeft:= ptrTAxisToolLeft^,
							TAxisToolCenter:= ptrTAxisToolCenter^,
							TAxisToolRight:=ptrTAxisToolRight^,
							TAxisToolFeeder:=ptrTAxisToolFeeder^,
							TAxisGrindFeeder:= ptrTAxisGrindFeeder^,
							xEnd=>ptrTFunction^.xEnd,
							xError=>ptrTFunction^.xError,
							iErrorNr=>ptrTFunction^.iErrorNr);
	END_IF;
	IF (iStationFunctionNr = 11) THEN
		(* AutoGeometry *)
		FBFctToolWorkingGeometry(	xMicroRodActive:= xMicroRodActive,
									xBeckhoffDriveActive:= xBeckhoffDriveActive,
									xSafetyCircuitOn:= xSafetyCircuitOn1 AND xSafetyCircuitOn2,
									T_ProcessImageData:= T_ProcessImageData,
									T_Standard:= T_Standard,
									xStart:= ptrTFunction^.xStart,
									xReset:=ptrTFunction^.xReset,
									xStop:= ptrTFunction^.xStop,
									xQuitErr:= ptrTFunction^.xQuitErr,
									xAbord:= ptrTFunction^.xAbord,
									TAxisToolLeft:= ptrTAxisToolLeft^,
									TAxisToolCenter:= ptrTAxisToolCenter^,
									TAxisToolRight:=ptrTAxisToolRight^,
									TAxisToolFeeder:=ptrTAxisToolFeeder^,
									TAxisGrindFeeder:= ptrTAxisGrindFeeder^,
									T_WorkTool:=TStation.T_WorkTool,
									xEnd=>ptrTFunction^.xEnd,
									xError=>ptrTFunction^.xError,
									iErrorNr=>ptrTFunction^.iErrorNr,
									bActivePartNumber=>bActivePartNumber,
									lrProcessToolFeederActualPosition=>lrProcessToolFeederActualPosition,
									lrProcessToolFeederSpeed=>lrProcessToolFeederSpeed,
									iCountDownPlungeCycle=>TStation.TControl.iCountDownPlungeCycle);
	END_IF;
	IF (iStationFunctionNr = 12) THEN
		(* AutoGroove *)
		FBFctToolWorkingGroove(		xMicroRodActive:= xMicroRodActive,
									xBeckhoffDriveActive:= xBeckhoffDriveActive,
									xSafetyCircuitOn:= xSafetyCircuitOn1 AND xSafetyCircuitOn2,
									xDoNotMoveGrindPosition:=T_ProcessImageData.T_AutoGroovePara.xBlockGrindFeeder,
									T_ProcessImageData:= T_ProcessImageData,
									T_Standard:= T_Standard,
									xStart:= ptrTFunction^.xStart,
									xReset:=ptrTFunction^.xReset,
									xStop:= ptrTFunction^.xStop,
									xQuitErr:= ptrTFunction^.xQuitErr,
									xAbord:= ptrTFunction^.xAbord,
									TAxisToolLeft:= ptrTAxisToolLeft^,
									TAxisToolCenter:= ptrTAxisToolCenter^,
									TAxisToolRight:=ptrTAxisToolRight^,
									TAxisToolFeeder:=ptrTAxisToolFeeder^,
									TAxisGrindFeeder:= ptrTAxisGrindFeeder^,
									T_WorkTool:=TStation.T_WorkTool,
									rStartPosAutoGrooveToolRotation:=TStation.rStartPosAutoGrooveToolRotation,
									xEnd=>ptrTFunction^.xEnd,
									xError=>ptrTFunction^.xError,
									iErrorNr=>ptrTFunction^.iErrorNr,
									bActivePartNumber=>bActivePartNumber,
									lrProcessToolFeederActualPosition=>lrProcessToolFeederActualPosition,
									lrProcessToolFeederSpeed=>lrProcessToolFeederSpeed);
	END_IF;
	IF (iStationFunctionNr = 13) THEN
		FBFctToolCalibration(			xMicroRodActive:= xMicroRodActive,
									xBeckhoffDriveActive:= xBeckhoffDriveActive,
									xSafetyCircuitOn:= xSafetyCircuitOn1 AND xSafetyCircuitOn2,
									T_ProcessImageData:= T_ProcessImageData,
									T_Standard:= T_Standard,
									xStart:= ptrTFunction^.xStart,
									xReset:=ptrTFunction^.xReset,
									xStop:= ptrTFunction^.xStop,
									xQuitErr:= ptrTFunction^.xQuitErr,
									xAbord:= ptrTFunction^.xAbord,
									TAxisToolLeft:= ptrTAxisToolLeft^,
									TAxisToolCenter:= ptrTAxisToolCenter^,
									TAxisToolRight:=ptrTAxisToolRight^,
									TAxisToolFeeder:=ptrTAxisToolFeeder^,
									TAxisGrindFeeder:= ptrTAxisGrindFeeder^,
									T_WorkTool:=TStation.T_WorkTool,
									xEnd=>ptrTFunction^.xEnd,
									xError=>ptrTFunction^.xError,
									iErrorNr=>ptrTFunction^.iErrorNr,
									lrProcessToolFeederActualPosition=>lrProcessToolFeederActualPosition,
									lrProcessToolFeederSpeed=>lrProcessToolFeederSpeed);
	END_IF;
	IF (iStationFunctionNr = 14) OR (iStationFunctionNr = 15) THEN
		FBFctToolFeedAbsRelPosition(		xMicroRodActive:= xMicroRodActive,
										xBeckhoffDriveActive:= xBeckhoffDriveActive,
										xSafetyCircuitOn:= xSafetyCircuitOn1 AND xSafetyCircuitOn2,
										iFunctionNr:= iStationFunctionNr,
										xStart:= ptrTFunction^.xStart,
										xReset:=ptrTFunction^.xReset,
										xStop:= ptrTFunction^.xStop,
										xQuitErr:= ptrTFunction^.xQuitErr,
										xAbord:= ptrTFunction^.xAbord,
										TAxisToolFeeder:= ptrTAxisToolFeeder^,
										xEnd=>ptrTFunction^.xEnd,
										xError=>ptrTFunction^.xError,
										iErrorNr=>ptrTFunction^.iErrorNr);
	END_IF;
	IF (iStationFunctionNr = 16) OR (iStationFunctionNr = 17) THEN
		FBFctSwitchOnOffPowerSupply(	xMicroRodActive:= xMicroRodActive,
									xBeckhoffDriveActive:= xBeckhoffDriveActive,
									xSafetyCircuitOn:= xSafetyCircuitOn1 AND xSafetyCircuitOn2,
									iFunctionNr:= iStationFunctionNr,
									xStart:= ptrTFunction^.xStart,
									xReset:=ptrTFunction^.xReset,
									xStop:= ptrTFunction^.xStop,
									xQuitErr:= ptrTFunction^.xQuitErr,
									xAbord:= ptrTFunction^.xAbord,
									TAxisToolLeft:= ptrTAxisToolLeft^,
									TAxisToolCenter:= ptrTAxisToolCenter^,
									TAxisToolRight:=ptrTAxisToolRight^,
									TAxisToolFeeder:=ptrTAxisToolFeeder^,
									TAxisGrindFeeder:= ptrTAxisGrindFeeder^,
									xEnd=>ptrTFunction^.xEnd,
									xError=>ptrTFunction^.xError,
									iErrorNr=>ptrTFunction^.iErrorNr);
	END_IF;
	IF (iStationFunctionNr = 18) THEN
		FBFctStopAxisMovement(	xMicroRodActive:= xMicroRodActive,
								xBeckhoffDriveActive:= xBeckhoffDriveActive,
								xSafetyCircuitOn:= xSafetyCircuitOn1 AND xSafetyCircuitOn2,
								T_ProcessImageData:= T_ProcessImageData,
								T_Standard:= T_Standard,
								xStart:= ptrTFunction^.xStart,
								xReset:=ptrTFunction^.xReset,
								xStop:= ptrTFunction^.xStop,
								xQuitErr:= ptrTFunction^.xQuitErr,
								xAbord:= ptrTFunction^.xAbord,
								TAxisToolLeft:= ptrTAxisToolLeft^,
								TAxisToolCenter:= ptrTAxisToolCenter^,
								TAxisToolRight:=ptrTAxisToolRight^,
								TAxisToolFeeder:=ptrTAxisToolFeeder^,
								TAxisGrindFeeder:= ptrTAxisGrindFeeder^,
								xEnd=>ptrTFunction^.xEnd,
								xError=>ptrTFunction^.xError,
								iErrorNr=>ptrTFunction^.iErrorNr);
	END_IF;
	IF (iStationFunctionNr = 19) THEN
		(* AutoGeometryMultiCycle*)
		FBFctToolWorkingGeometryMultiCycle(	xMicroRodActive:= xMicroRodActive,
											xBeckhoffDriveActive:= xBeckhoffDriveActive,
											xSafetyCircuitOn:= xSafetyCircuitOn1 AND xSafetyCircuitOn2,
											T_ProcessImageData:= T_ProcessImageData,
											T_Standard:= T_Standard,
											xStart:= ptrTFunction^.xStart,
											xReset:=ptrTFunction^.xReset,
											xStop:= ptrTFunction^.xStop,
											xQuitErr:= ptrTFunction^.xQuitErr,
											xAbord:= ptrTFunction^.xAbord,
											TAxisToolLeft:= ptrTAxisToolLeft^,
											TAxisToolCenter:= ptrTAxisToolCenter^,
											TAxisToolRight:=ptrTAxisToolRight^,
											TAxisToolFeeder:=ptrTAxisToolFeeder^,
											TAxisGrindFeeder:= ptrTAxisGrindFeeder^,
											T_WorkTool:=TStation.T_WorkTool,
											xEnd=>ptrTFunction^.xEnd,
											xError=>ptrTFunction^.xError,
											iErrorNr=>ptrTFunction^.iErrorNr,
											bActivePartNumber=>bActivePartNumber,
											lrProcessToolFeederActualPosition=>lrProcessToolFeederActualPosition,
											lrProcessToolFeederSpeed=>lrProcessToolFeederSpeed,
											iCountDownPlungeCycle=>TStation.TControl.iCountDownPlungeCycle);
	END_IF;
	(* 17.11.2010: KFS 	{	*)
	IF (iStationFunctionNr = 20) THEN
		FBFctToolFeedMaxLenReference(	xMicroRodActive:= xMicroRodActive,
										xBeckhoffDriveActive:= xBeckhoffDriveActive,
										xSafetyCircuitOn:= xSafetyCircuitOn1 AND xSafetyCircuitOn2,
										T_Standard:= T_Standard,
										xStart:= ptrTFunction^.xStart,
										xReset:=ptrTFunction^.xReset,
										xStop:= ptrTFunction^.xStop,
										xQuitErr:= ptrTFunction^.xQuitErr,
										xAbord:= ptrTFunction^.xAbord,
										TAxisToolFeeder:= ptrTAxisToolFeeder^,
										xEnd=>ptrTFunction^.xEnd,
										xError=>ptrTFunction^.xError,
										iErrorNr=>ptrTFunction^.iErrorNr);
	END_IF;
	(* 17.11.2010: KFS 	{	*)
END_IF;
(******************************************************************************************************************************************)
(****************************				         Init / Reset Hardware                                                 *****************************)
(******************************************************************************************************************************************)
IF xSetEnd THEN
	xStationError:=FALSE;
	xInitError:=FALSE;
	xInitStart:=FALSE;
	xInitStop:=FALSE;
	xInitStep:=FALSE;
	xSetEnd:=FALSE;
	xTmpStart:=FALSE;
	TStation.TControl.xEnd:=TRUE;
	TStation.TControl.xStart:=FALSE;
	TStation.TControl.xStop:=FALSE;
	TStation.TControl.xAbord:=FALSE;
	IF NOT(xDontDeleteErrorFlag) THEN
		TStation.TControl.xError:=FALSE;
		TStation.TControl.diErrorNr:=0;
	END_IF;
	xDontDeleteErrorFlag:=FALSE;
	xStartFunction:=FALSE;
	iStepError:=100;
	xStepError:=FALSE;
	xTmpStationError:=FALSE;
	xChkConfigStation:=FALSE;
	diErrorNumber:=0;
	xSetError:=FALSE;
	xReadyToQuitErr:=FALSE;
END_IF;
(*03.03.2017: KFS { *)
IF T_StartUp.T_State.xCompleted THEN
	IF ptrTCylToolLeftActive^.T_CtrleCyl.T_Standard.xActivOn AND ptrTAxisToolLeft^.T_CtrleSingle.xPower
	     AND NOT(ptrTAxisToolLeft^.T_CtrleSingle.xExecute) AND ptrTAxisToolLeft^.T_CtrleSingle.xDone THEN
		ptrTAxisToolLeft^.T_CtrleSingle.iFunction:=4;
		ptrTAxisToolLeft^.T_CtrleSingle.xExecute:=TRUE;
	END_IF;
	IF ptrTCylToolRightActive^.T_CtrleCyl.T_Standard.xActivOn AND ptrTAxisToolRight^.T_CtrleSingle.xPower
	     AND NOT(ptrTAxisToolRight^.T_CtrleSingle.xExecute) AND ptrTAxisToolRight^.T_CtrleSingle.xDone THEN
		ptrTAxisToolRight^.T_CtrleSingle.iFunction:=4;
		ptrTAxisToolRight^.T_CtrleSingle.xExecute:=TRUE;
	END_IF;
END_IF;
(*03.03.2017: KFS } *)
END_FUNCTION_BLOCK

(* POU PRG_STATION_LAYER3/FB_STATIONEN/FB_FUNCTION/FB_FctToolRotationTorqueStart, ST *)
FUNCTION_BLOCK FB_FctToolRotationTorqueStart
VAR_INPUT
	xMicroRodActive: BOOL;		(* choice of the machine MicroWire or MicroRod *)
	xBeckhoffDriveActive: BOOL;	(* choice of the axis Beckhoff or EcoStep *)
	xSafetyCircuitOn:BOOL;			(* state of the safety circuit-->TRUE=Machine current ON, FALSE=Machine current OFF *)
END_VAR
VAR_IN_OUT
	xStart : BOOL;					(* start the function *)
	xReset : BOOL;				(* reset the function *)
	xStop : BOOL;					(* stop the active function *)
	xQuitErr : BOOL;				(* quit the error caused of the active function *)
	xAbord : BOOL;				(* abord the active function *)
	TAxisToolLeft:ST_AXIS;		(* data structure for the ToolLeft axis *)
	TAxisToolCenter:ST_AXIS;		(* data structure for the ToolCenter axis *)
	TAxisToolRight:ST_AXIS;		(* data structure for the ToolRight axis *)
	TAxisToolFeeder:ST_AXIS;		(* data structure for the ToolFeeder axis *)
END_VAR
VAR_OUTPUT
	xEnd : BOOL;					(* state of the function if a active function is ended *)
	xError : BOOL;					(* state of the function if a active function caused an error *)
	iErrorNr : INT;					(* state of the function if a active function caused an error, in this case give the error number *)
END_VAR
VAR
	xHardwareError: BOOL := FALSE;
	xInitError: BOOL := FALSE;
	iStepError: INT := 0;
	xStartMainCtr: BOOL := FALSE;
	xStartMainPrc: BOOL := FALSE;
	xInitMainCtr: BOOL := FALSE;
	iStepPrc: INT := 0;
	xSetEnd: BOOL := FALSE;
	xInitStep: BOOL := FALSE;
	xFreeze: BOOL := FALSE;
	iTmpErrorNr:INT:=0;
	xTmpInit:BOOL;
	iTmp:INT;
	xTmp: BOOL;
	TONWaitStop: TON;
END_VAR
(****************************************************************************************************************************************************)
(***********                                      This Functionblock define the function for start the toolrotation                                                    ************)
(****************************************************************************************************************************************************)

(******************************************************************************************************************************************)
(****************************				           Reset Function Part                                                 *****************************)
(******************************************************************************************************************************************)
IF xReset AND NOT(xSetEnd) THEN
	xEnd:=FALSE;
	xSetEnd:=TRUE;
END_IF;
(******************************************************************************************************************************************)
(****************************				              Error Controlling Part                                            *****************************)
(******************************************************************************************************************************************)
IF (xHardwareError OR ((TAxisToolLeft.T_CtrleSingle.xErr OR (TAxisToolCenter.T_CtrleSingle.xErr AND xMicroRodActive) OR TAxisToolRight.T_CtrleSingle.xErr OR (TAxisToolFeeder.T_CtrleSingle.xErr AND NOT(xMicroRodActive))) AND xStartMainPrc)) AND NOT(xSetEnd) THEN
	IF NOT(TAxisToolLeft.T_CtrleSingle.xExecute) AND ((NOT(TAxisToolCenter.T_CtrleSingle.xExecute) AND xMicroRodActive) OR NOT(xMicroRodActive)) AND NOT(TAxisToolRight.T_CtrleSingle.xExecute) AND ((NOT(TAxisToolFeeder.T_CtrleSingle.xExecute) AND NOT(xMicroRodActive)) OR xMicroRodActive) THEN
		IF NOT(xInitError) THEN
			iStepError:=100;
			xInitError:=TRUE;
			IF xHardwareError THEN
				iErrorNr:=iTmpErrorNr;
			ELSE
				xHardwareError:=TRUE;	(* Hardware Error *)
			END_IF;
		END_IF;
		CASE iStepError OF
			100:	iStepError:=0;
				xError:=TRUE;
		END_CASE;
		IF xQuitErr THEN
			xSetEnd:=TRUE;
		END_IF;
	END_IF;
END_IF;
(******************************************************************************************************************************************)
(****************************				              Main Controlling Part                                            *****************************)
(******************************************************************************************************************************************)
IF (xStart OR xStartMainCtr) AND NOT(xSetEnd) AND NOT(xHardwareError) THEN
	IF NOT (xInitMainCtr) THEN
		iTmpErrorNr:=0;
		iStepPrc:=100;
		xInitMainCtr:=TRUE;
		xStartMainCtr:=TRUE;
		xStart:=FALSE;
		xEnd:=FALSE;
		xAbord:=FALSE;
		xTmpInit:=FALSE;
	END_IF;
	IF xStop AND NOT(xTmpInit) THEN
		xTmpInit:=TRUE;
		iTmp:=100;
		RETURN;
	END_IF;
	IF xFreeze THEN
		IF xStart AND NOT(xAbord) THEN
			xFreeze:=FALSE;
			xStart:=FALSE;
		END_IF;
		IF xAbord THEN
			xAbord:=FALSE;
			xFreeze:=FALSE;
			xStart:=FALSE;
			xSetEnd:=TRUE;
		END_IF;
		RETURN;
	END_IF;
	IF NOT(xStartMainPrc) AND NOT(xSetEnd) THEN
		xStartMainPrc:=TRUE;
	END_IF;
END_IF;
(******************************************************************************************************************************************)
(****************************				             immediate Stop Part                                              *****************************)
(******************************************************************************************************************************************)
IF xTmpInit AND NOT(xSetEnd) THEN
	IF NOT(xSafetyCircuitOn) THEN
		xTmpInit:=FALSE;
		iTmp:=100;
		xSetEnd:=TRUE;
		RETURN;
	END_IF;
	CASE iTmp OF
		100:	IF TAxisToolLeft.T_CtrleSingle.xDone OR (TAxisToolCenter.T_CtrleSingle.xDone AND xMicroRodActive) OR TAxisToolRight.T_CtrleSingle.xDone OR (TAxisToolFeeder.T_CtrleSingle.xDone AND NOT(xMicroRodActive)) THEN
				TAxisToolLeft.T_CtrleSingle.iFunction:=5;
				TAxisToolLeft.T_CtrleSingle.xExecute:=TRUE;
				iTmp:=200;
			END_IF;
			RETURN;
		200:	IF NOT(TAxisToolLeft.T_CtrleSingle.xExecute) AND TAxisToolLeft.T_CtrleSingle.xDone THEN
				iTmp:=300;
				TONWaitStop(IN:=FALSE);
			END_IF;
			RETURN;
		300:	xTmp:=	((UINT_TO_WORD(TAxisToolRight.T_TxPdoParameter.uiStatusWord) AND 16#1000) = 16#1000) AND
					((((UINT_TO_WORD(TAxisToolCenter.T_TxPdoParameter.uiStatusWord) AND 16#1000) = 16#1000) AND xMicroRodActive) OR NOT(xMicroRodActive)) AND
					((((UINT_TO_WORD(TAxisToolFeeder.T_TxPdoParameter.uiStatusWord) AND 16#1000) = 16#1000) AND NOT(xMicroRodActive)) OR xMicroRodActive);
			TONWaitStop(IN:=TRUE,PT:=T#1000ms);
			IF TONWaitStop.Q AND xTmp THEN
				TONWaitStop(IN:=FALSE);
				iTmp:=400;
			END_IF;
			RETURN;
		400:	IF xMicroRodActive THEN
				IF TAxisToolCenter.T_CtrleSingle.xSlave THEN
					TAxisToolCenter.T_CtrleSingle.iFunction:=25;
					TAxisToolCenter.T_CtrleSingle.xExecute:=TRUE;
				END_IF;
			END_IF;
			IF TAxisToolRight.T_CtrleSingle.xSlave THEN
				TAxisToolRight.T_CtrleSingle.iFunction:=25;
				TAxisToolRight.T_CtrleSingle.xExecute:=TRUE;
			END_IF;
			IF NOT(xMicroRodActive) THEN
				IF TAxisToolFeeder.T_CtrleSingle.xSlave THEN
					TAxisToolFeeder.T_CtrleSingle.iFunction:=25;
					TAxisToolFeeder.T_CtrleSingle.xExecute:=TRUE;
				END_IF;
			END_IF;
			iTmp:=500;
			RETURN;
		500:	IF ((NOT(TAxisToolCenter.T_CtrleSingle.xExecute) AND TAxisToolCenter.T_CtrleSingle.xDone AND xMicroRodActive) OR NOT(xMicroRodActive)) AND
			    NOT(TAxisToolRight.T_CtrleSingle.xExecute) AND TAxisToolRight.T_CtrleSingle.xDone AND
			    ((NOT(TAxisToolFeeder.T_CtrleSingle.xExecute) AND TAxisToolFeeder.T_CtrleSingle.xDone AND NOT(xMicroRodActive)) OR xMicroRodActive) THEN
				xTmpInit:=FALSE;
				iTmp:=100;
				xSetEnd:=TRUE;
			END_IF;
			RETURN;
	END_CASE;
END_IF;
(******************************************************************************************************************************************)
(****************************				             Main Procedure Part                                             *****************************)
(******************************************************************************************************************************************)
IF xStartMainPrc AND NOT(xSetEnd) AND NOT(xHardwareError) THEN
	CASE iStepPrc OF
		100:	IF NOT(xInitStep) THEN
				xInitStep:=TRUE;
				IF NOT(TAxisToolLeft.T_CtrleSingle.xDone) OR (NOT(TAxisToolCenter.T_CtrleSingle.xDone) AND xMicroRodActive) OR NOT(TAxisToolRight.T_CtrleSingle.xDone) OR (NOT(TAxisToolFeeder.T_CtrleSingle.xDone) AND NOT(xMicroRodActive)) THEN
					xHardwareError:=TRUE;
					iTmpErrorNr:=1;
					RETURN;
				END_IF;
				IF NOT(TAxisToolLeft.T_CtrleSingle.xPower) THEN
					TAxisToolLeft.T_CtrleSingle.iFunction:=3;
					TAxisToolLeft.T_CtrleSingle.xExecute:=TRUE;
				END_IF;
				IF xMicroRodActive THEN
					IF NOT(TAxisToolCenter.T_CtrleSingle.xPower) THEN
						TAxisToolCenter.T_CtrleSingle.iFunction:=3;
						TAxisToolCenter.T_CtrleSingle.xExecute:=TRUE;
					END_IF;
				END_IF;
				IF NOT(TAxisToolRight.T_CtrleSingle.xPower) THEN
					TAxisToolRight.T_CtrleSingle.iFunction:=3;
					TAxisToolRight.T_CtrleSingle.xExecute:=TRUE;
				END_IF;
				IF NOT(xMicroRodActive) THEN
					IF NOT(TAxisToolFeeder.T_CtrleSingle.xPower) THEN
						TAxisToolFeeder.T_CtrleSingle.iFunction:=3;
						TAxisToolFeeder.T_CtrleSingle.xExecute:=TRUE;
					END_IF;
				END_IF;
			END_IF;
			IF NOT(TAxisToolLeft.T_CtrleSingle.xExecute) AND TAxisToolLeft.T_CtrleSingle.xDone AND
			    ((NOT(TAxisToolCenter.T_CtrleSingle.xExecute) AND TAxisToolCenter.T_CtrleSingle.xDone AND xMicroRodActive) OR NOT(xMicroRodActive)) AND
			    NOT(TAxisToolRight.T_CtrleSingle.xExecute) AND TAxisToolRight.T_CtrleSingle.xDone AND
			    ((NOT(TAxisToolFeeder.T_CtrleSingle.xExecute) AND TAxisToolFeeder.T_CtrleSingle.xDone AND NOT(xMicroRodActive)) OR xMicroRodActive) THEN
				xStartMainPrc:=FALSE;
				xInitStep:=FALSE;
				iStepPrc:=200;
			END_IF;
		200:	IF NOT(xInitStep) THEN
				xInitStep:=TRUE;
				IF xMicroRodActive THEN
					IF NOT(TAxisToolCenter.T_CtrleSingle.xSlave) THEN
						TAxisToolCenter.T_CtrleSingle.iFunction:=25;
						TAxisToolCenter.T_CtrleSingle.xExecute:=TRUE;
					END_IF;
				END_IF;
				IF NOT(TAxisToolRight.T_CtrleSingle.xSlave) THEN
					TAxisToolRight.T_CtrleSingle.iFunction:=25;
					TAxisToolRight.T_CtrleSingle.xExecute:=TRUE;
				END_IF;
				IF NOT(xMicroRodActive) THEN
					IF NOT(TAxisToolFeeder.T_CtrleSingle.xSlave) THEN
						TAxisToolFeeder.T_CtrleSingle.iFunction:=25;
						TAxisToolFeeder.T_CtrleSingle.xExecute:=TRUE;
					END_IF;
				END_IF;
			END_IF;
			IF ((NOT(TAxisToolCenter.T_CtrleSingle.xExecute) AND TAxisToolCenter.T_CtrleSingle.xDone AND xMicroRodActive) OR NOT(xMicroRodActive)) AND
			    NOT(TAxisToolRight.T_CtrleSingle.xExecute) AND TAxisToolRight.T_CtrleSingle.xDone AND
			    ((NOT(TAxisToolFeeder.T_CtrleSingle.xExecute) AND TAxisToolFeeder.T_CtrleSingle.xDone AND NOT(xMicroRodActive)) OR xMicroRodActive) THEN
				xStartMainPrc:=FALSE;
				xInitStep:=FALSE;
				iStepPrc:=300;
			END_IF;
		300:	IF NOT(xInitStep) THEN
				xInitStep:=TRUE;
				TAxisToolLeft.T_CtrleSingle.iFunction:=6;
				TAxisToolLeft.T_CtrleSingle.xExecute:=TRUE;
			END_IF;
			IF NOT(TAxisToolLeft.T_CtrleSingle.xExecute) AND TAxisToolLeft.T_CtrleSingle.xDone THEN
				xStartMainPrc:=FALSE;
				xInitStep:=FALSE;
				iStepPrc:=0;
				xSetEnd:=TRUE;
			END_IF;
	END_CASE;
END_IF;
(******************************************************************************************************************************************)
(****************************				           Parallel Procedure Part                                          *****************************)
(******************************************************************************************************************************************)

(******************************************************************************************************************************************)
(****************************				             	Init / Reset Part                                                   *****************************)
(******************************************************************************************************************************************)
IF xSetEnd THEN
	xEnd:=TRUE;
	xInitStep:=FALSE;
	xSetEnd:=FALSE;
	xStop:=FALSE;
	xStartMainPrc:=FALSE;
	xInitMainCtr:=FALSE;
	xStartMainCtr:=FALSE;
	xStart:=FALSE;
	xHardwareError:=FALSE;
	xQuitErr:=FALSE;
	xError:=FALSE;
	iErrorNr:=0;
	xInitError:=FALSE;
	xFreeze:=FALSE;
	xAbord:=FALSE;
	xReset:=FALSE;
END_IF;
END_FUNCTION_BLOCK

(* POU PRG_STATION_LAYER3/FB_STATIONEN/FB_FUNCTION/FB_FctToolRotationTorqueStop, ST *)
FUNCTION_BLOCK FB_FctToolRotationTorqueStop
VAR_INPUT
	xMicroRodActive: BOOL;		(* choice of the machine MicroWire or MicroRod *)
	xBeckhoffDriveActive: BOOL;	(* choice of the axis Beckhoff or EcoStep *)
	xSafetyCircuitOn:BOOL;			(* state of the safety circuit-->TRUE=Machine current ON, FALSE=Machine current OFF *)
END_VAR
VAR_IN_OUT
	xStart : BOOL;					(* start the function *)
	xReset : BOOL;				(* reset the function *)
	xStop : BOOL;					(* stop the active function *)
	xQuitErr : BOOL;				(* quit the error caused of the active function *)
	xAbord : BOOL;				(* abord the active function *)
	TAxisToolLeft:ST_AXIS;		(* data structure for the ToolLeft axis *)
	TAxisToolCenter:ST_AXIS;		(* data structure for the ToolCenter axis *)
	TAxisToolRight:ST_AXIS;		(* data structure for the ToolRight axis *)
	TAxisToolFeeder:ST_AXIS;		(* data structure for the ToolFeeder axis *)
END_VAR
VAR_OUTPUT
	xEnd : BOOL;					(* state of the function if a active function is ended *)
	xError : BOOL;					(* state of the function if a active function caused an error *)
	iErrorNr : INT;					(* state of the function if a active function caused an error, in this case give the error number *)
END_VAR
VAR
	xHardwareError: BOOL := FALSE;
	xInitError: BOOL := FALSE;
	iStepError: INT := 0;
	xStartMainCtr: BOOL := FALSE;
	xStartMainPrc: BOOL := FALSE;
	xInitMainCtr: BOOL := FALSE;
	iStepPrc: INT := 0;
	xSetEnd: BOOL := FALSE;
	xInitStep: BOOL := FALSE;
	xFreeze: BOOL := FALSE;
	iTmpErrorNr:INT:=0;
	xTmpInit:BOOL;
	iTmp:INT;
	xTmp: BOOL;
	TONWaitStop: TON;
END_VAR
(****************************************************************************************************************************************************)
(***********                                      This Functionblock define the function for stop the toolrotation                                                    ************)
(****************************************************************************************************************************************************)

(******************************************************************************************************************************************)
(****************************				           Reset Function Part                                                 *****************************)
(******************************************************************************************************************************************)
IF xReset AND NOT(xSetEnd) THEN
	xEnd:=FALSE;
	xSetEnd:=TRUE;
END_IF;
(******************************************************************************************************************************************)
(****************************				              Error Controlling Part                                            *****************************)
(******************************************************************************************************************************************)
IF (xHardwareError OR ((TAxisToolLeft.T_CtrleSingle.xErr OR (TAxisToolCenter.T_CtrleSingle.xErr AND xMicroRodActive) OR TAxisToolRight.T_CtrleSingle.xErr OR (TAxisToolFeeder.T_CtrleSingle.xErr AND NOT(xMicroRodActive))) AND xStartMainPrc)) AND NOT(xSetEnd) THEN
	IF NOT(TAxisToolLeft.T_CtrleSingle.xExecute) AND ((NOT(TAxisToolCenter.T_CtrleSingle.xExecute) AND xMicroRodActive) OR NOT(xMicroRodActive)) AND NOT(TAxisToolRight.T_CtrleSingle.xExecute) AND ((NOT(TAxisToolFeeder.T_CtrleSingle.xExecute) AND NOT(xMicroRodActive)) OR xMicroRodActive) THEN
		IF NOT(xInitError) THEN
			iStepError:=100;
			xInitError:=TRUE;
			IF xHardwareError THEN
				iErrorNr:=iTmpErrorNr;
			ELSE
				xHardwareError:=TRUE;	(* Hardware Error *)
			END_IF;
		END_IF;
		CASE iStepError OF
			100:	iStepError:=0;
				xError:=TRUE;
		END_CASE;
		IF xQuitErr THEN
			xSetEnd:=TRUE;
		END_IF;
	END_IF;
END_IF;
(******************************************************************************************************************************************)
(****************************				              Main Controlling Part                                            *****************************)
(******************************************************************************************************************************************)
IF (xStart OR xStartMainCtr) AND NOT(xSetEnd) AND NOT(xHardwareError) THEN
	IF NOT (xInitMainCtr) THEN
		iTmpErrorNr:=0;
		iStepPrc:=100;
		xInitMainCtr:=TRUE;
		xStartMainCtr:=TRUE;
		xStart:=FALSE;
		xEnd:=FALSE;
		xAbord:=FALSE;
		xTmpInit:=FALSE;
	END_IF;
	IF xStop AND NOT(xTmpInit) THEN
		xTmpInit:=TRUE;
		iTmp:=100;
		RETURN;
	END_IF;
	IF xFreeze THEN
		IF xStart AND NOT(xAbord) THEN
			xFreeze:=FALSE;
			xStart:=FALSE;
		END_IF;
		IF xAbord THEN
			xAbord:=FALSE;
			xFreeze:=FALSE;
			xStart:=FALSE;
			xSetEnd:=TRUE;
		END_IF;
		RETURN;
	END_IF;
	IF NOT(xStartMainPrc) AND NOT(xSetEnd) THEN
		xStartMainPrc:=TRUE;
	END_IF;
END_IF;
(******************************************************************************************************************************************)
(****************************				             immediate Stop Part                                              *****************************)
(******************************************************************************************************************************************)
IF xTmpInit AND NOT(xSetEnd) THEN
	IF NOT(xSafetyCircuitOn) THEN
		xTmpInit:=FALSE;
		iTmp:=100;
		xSetEnd:=TRUE;
		RETURN;
	END_IF;
	CASE iTmp OF
		(* No immediately stopping *)
		100:	xTmpInit:=FALSE;
			iTmp:=100;
	END_CASE;
END_IF;
(******************************************************************************************************************************************)
(****************************				             Main Procedure Part                                             *****************************)
(******************************************************************************************************************************************)
IF xStartMainPrc AND NOT(xSetEnd) AND NOT(xHardwareError) THEN
	CASE iStepPrc OF
		100:	IF NOT(xInitStep) THEN
				xInitStep:=TRUE;
				IF NOT(TAxisToolLeft.T_CtrleSingle.xDone) OR (NOT(TAxisToolCenter.T_CtrleSingle.xDone) AND xMicroRodActive) OR NOT(TAxisToolRight.T_CtrleSingle.xDone) OR (NOT(TAxisToolFeeder.T_CtrleSingle.xDone) AND NOT(xMicroRodActive)) THEN
					xHardwareError:=TRUE;
					iTmpErrorNr:=1;
					RETURN;
				END_IF;
				TAxisToolLeft.T_CtrleSingle.iFunction:=5;
				TAxisToolLeft.T_CtrleSingle.xExecute:=TRUE;
			END_IF;
			IF NOT(TAxisToolLeft.T_CtrleSingle.xExecute) AND TAxisToolLeft.T_CtrleSingle.xDone THEN
				xStartMainPrc:=FALSE;
				xInitStep:=FALSE;
				iStepPrc:=199;
			END_IF;
		199:	xTmp:=	((UINT_TO_WORD(TAxisToolRight.T_TxPdoParameter.uiStatusWord) AND 16#1000) = 16#1000) AND
					((((UINT_TO_WORD(TAxisToolCenter.T_TxPdoParameter.uiStatusWord) AND 16#1000) = 16#1000) AND xMicroRodActive) OR NOT(xMicroRodActive)) AND
					((((UINT_TO_WORD(TAxisToolFeeder.T_TxPdoParameter.uiStatusWord) AND 16#1000) = 16#1000) AND NOT(xMicroRodActive)) OR xMicroRodActive);
			IF NOT(xInitStep) THEN
				xInitStep:=TRUE;
				TONWaitStop(IN:=FALSE);
			END_IF;
			TONWaitStop(IN:=TRUE,PT:=T#1000ms);
			IF TONWaitStop.Q AND xTmp THEN
				TONWaitStop(IN:=FALSE);
				xStartMainPrc:=FALSE;
				xInitStep:=FALSE;
				iStepPrc:=200;
			END_IF;
		200:	IF NOT(xInitStep) THEN
				xInitStep:=TRUE;
				IF xMicroRodActive THEN
					IF TAxisToolCenter.T_CtrleSingle.xSlave THEN
						TAxisToolCenter.T_CtrleSingle.iFunction:=25;
						TAxisToolCenter.T_CtrleSingle.xExecute:=TRUE;
					END_IF;
				END_IF;
				IF TAxisToolRight.T_CtrleSingle.xSlave THEN
					TAxisToolRight.T_CtrleSingle.iFunction:=25;
					TAxisToolRight.T_CtrleSingle.xExecute:=TRUE;
				END_IF;
				IF NOT(xMicroRodActive) THEN
					IF TAxisToolFeeder.T_CtrleSingle.xSlave THEN
						TAxisToolFeeder.T_CtrleSingle.iFunction:=25;
						TAxisToolFeeder.T_CtrleSingle.xExecute:=TRUE;
					END_IF;
				END_IF;
			END_IF;
			IF ((NOT(TAxisToolCenter.T_CtrleSingle.xExecute) AND TAxisToolCenter.T_CtrleSingle.xDone AND xMicroRodActive) OR NOT(xMicroRodActive)) AND
			    NOT(TAxisToolRight.T_CtrleSingle.xExecute) AND TAxisToolRight.T_CtrleSingle.xDone AND
			    ((NOT(TAxisToolFeeder.T_CtrleSingle.xExecute) AND TAxisToolFeeder.T_CtrleSingle.xDone AND NOT(xMicroRodActive)) OR xMicroRodActive) THEN
				xStartMainPrc:=FALSE;
				xInitStep:=FALSE;
				iStepPrc:=0;
				xSetEnd:=TRUE;
			END_IF;
	END_CASE;
END_IF;
(******************************************************************************************************************************************)
(****************************				           Parallel Procedure Part                                          *****************************)
(******************************************************************************************************************************************)

(******************************************************************************************************************************************)
(****************************				             	Init / Reset Part                                                   *****************************)
(******************************************************************************************************************************************)
IF xSetEnd THEN
	xEnd:=TRUE;
	xInitStep:=FALSE;
	xSetEnd:=FALSE;
	xStop:=FALSE;
	xStartMainPrc:=FALSE;
	xInitMainCtr:=FALSE;
	xStartMainCtr:=FALSE;
	xStart:=FALSE;
	xHardwareError:=FALSE;
	xQuitErr:=FALSE;
	xError:=FALSE;
	iErrorNr:=0;
	xInitError:=FALSE;
	xFreeze:=FALSE;
	xAbord:=FALSE;
	xReset:=FALSE;
END_IF;
END_FUNCTION_BLOCK

(* POU PRG_STATION_LAYER3/FB_STATIONEN/FB_FUNCTION/FB_FctGrindFeedAbsRelPosition, ST *)
FUNCTION_BLOCK FB_FctGrindFeedAbsRelPosition
VAR_INPUT
	xMicroRodActive: BOOL;		(* choice of the machine MicroWire or MicroRod *)
	xBeckhoffDriveActive: BOOL;	(* choice of the axis Beckhoff or EcoStep *)
	xSafetyCircuitOn:BOOL;			(* state of the safety circuit-->TRUE=Machine current ON, FALSE=Machine current OFF *)
	iFunctionNr:INT;				(* state of the called function number-->4=move axis absolut, 5=move axis relative *)
END_VAR
VAR_IN_OUT
	xStart : BOOL;					(* start the function *)
	xReset : BOOL;				(* reset the function *)
	xStop : BOOL;					(* stop the active function *)
	xQuitErr : BOOL;				(* quit the error caused of the active function *)
	xAbord : BOOL;				(* abord the active function *)
	TAxisGrindFeeder:ST_AXIS;	(* data structure for the GrindFeeder axis *)
END_VAR
VAR_OUTPUT
	xEnd : BOOL;					(* state of the function if a active function is ended *)
	xError : BOOL;					(* state of the function if a active function caused an error *)
	iErrorNr : INT;					(* state of the function if a active function caused an error, in this case give the error number *)
END_VAR
VAR
	xHardwareError: BOOL := FALSE;
	xInitError: BOOL := FALSE;
	iStepError: INT := 0;
	xStartMainCtr: BOOL := FALSE;
	xStartMainPrc: BOOL := FALSE;
	xInitMainCtr: BOOL := FALSE;
	iStepPrc: INT := 0;
	xSetEnd: BOOL := FALSE;
	xInitStep: BOOL := FALSE;
	xFreeze: BOOL := FALSE;
	iTmpErrorNr:INT:=0;
	xTmpInit:BOOL;
	iTmp:INT;
END_VAR
(****************************************************************************************************************************************************)
(***********       This Functionblock define the function for set the GrindFeeder Axis to the relative or absolut position       ************)
(****************************************************************************************************************************************************)

